# B&R Automation Studio project AS
Automation Studio 4.2.4.149

## Configuration Config1

CPU 5PC800.B945-02, AutomationRuntime A4.26, Build 4.1.2, Vc V4.26.0

### Cpu.per - 5PC800_B945_02/Cpu.per
```iecst
VAR_CONFIG
	gRecCfg AT %M0; (* *)
END_VAR
```

### cncSpindle.mpspindle - 5PC800_B945_02/mapp/cncSpindle.mpspindle
```
Element Spindle_MpLink (Type=mpspindle)
  AxisConfiguration = AxisWithConfiguration
    Axis:
      MeasurementResolution = 0.001
      MovementLimits:
        VelocityPositive = 360000
        VelocityNegative = 360000
        Acceleration = 36000
        Deceleration = 36000
        JerkTime = 0.01
    Drive:
      Controller:
        LoopFilters:
          [0]
          [1]
          [2]
  Alarms = MpAlarmX
```

### deltaCtrl.mpdelta4axis - 5PC800_B945_02/mapp/deltaCtrl.mpdelta4axis
```
Element Delta_MpLink (Type=mpdelta4axis)
  Linking:
    Subnodes:
      JointQ1 = Axis_Delta_Joint_Q1_MpLink
      JointQ2 = Axis_Delta_Joint_Q2_MpLink
      JointQ3 = Axis_Delta_Joint_Q3_MpLink
      Rotary = Axis_Delta_Joint_Q4_MpLink
  Robot:
    Mechanics:
      BasePosition:
        Z = 938.87
      ArmLinkPoint:
        [0]:
          Radius = 200
        [1]:
          Angle = 120
          Radius = 200
        [2]:
          Angle = 240
          Radius = 200
      ArmLength:
        [0]:
          UpperArm = 350
          LowerArm = 800
        [1]:
          UpperArm = 350
          LowerArm = 800
        [2]:
          UpperArm = 350
          LowerArm = 800
      TCPLinkPoint:
        [0]:
          Radius = 45
        [1]:
          Radius = 45
        [2]:
          Radius = 45
    Joint:
      [0]:
        NegativeMoveLimit = -150
        PositiveMoveLimit = 970
        UseTRFLimits = FALSE
      [1]:
        NegativeMoveLimit = -150
        PositiveMoveLimit = 970
        UseTRFLimits = FALSE
      [2]:
        NegativeMoveLimit = -150
        PositiveMoveLimit = 970
        UseTRFLimits = FALSE
    Rotary:
      UseTRFLimits = FALSE
    WorkspaceMonitoring:
      ProtectedBlock:
        [0]
        [1]
        [2]
        [3]
        [4]
      ProtectedHalfSpace:
        [0]
        [1]
        [2]
        [3]
        [4]
  Alarms = MpAlarmX
```

## Configuration Config_MpView

CPU 5PC800.B945-02, AutomationRuntime A4.26, Build 4.1.2, Vc V4.26.0, Safety 0.0

### Arnc0cfg.ncc - 5PC800_B945_02/Motion/Arnc0cfg.ncc
```
NcConfiguration (Version=3.14.3, NcSwId=Arnc0)
  ARNC0CFG_typ:
    sampling_rate = 2000
    cnt_nettrc_rec_drive = 150
    bufsize_sys_trace = 16#00005000
    enable_mp_log = Yes
    tc_nc_man_task = Cyclic #1
    bg_load = 1
    glob_pv_as_ncobject = No
```

### AlarmXCore.mpalarmxcore - 5PC800_B945_02/mapp/AlarmXCore.mpalarmxcore
```
Element MpLink_AlarmControl (Type=mpalarmxcore)
  mapp.AlarmX.Core:
    Mapping:
      [0]:
        Alarm = exampleAlarm
        [0] = Reaction
          Name = exampleReaction
    Default:
      [0] = Reaction
  mapp.AlarmX.Core.Configuration:
    [0]:
      Name = exampleAlarm
      Message = {$alarm/txtExampleAlarm}
      Code = 123456
  mapp.AlarmX.Core.Snippets:
    [0]:
      Key = exampleSnippet
      Value:
        PV = ::AlarmX:loc.val_float
```

### Energy.mpenergycore - 5PC800_B945_02/mapp/Energy.mpenergycore
```
Element Energy_MpLink (Type=mpenergycore)
  Alarms = MpAlarmX
```

### RecCfg.mprecipecsv - 5PC800_B945_02/mapp/RecCfg.mprecipecsv
```
Element Recipe_CSV_MpLink (Type=mprecipecsv)
  mapp.Recipe.Csv:
    Format:
      DecimalMark = .
  Alarms = MpAlarmX
Element Config_CSV_MpLink (Type=mprecipecsv)
  mapp.Recipe.Csv:
    Format:
      DecimalMark = .
  Alarms = MpAlarmX
```

### cncAxes.mpaxisbasic - 5PC800_B945_02/mapp/cncAxes.mpaxisbasic
```
Element Axis_CNC_Z_MpLink (Type=mpaxisbasic)
  AxisConfiguration = AxisWithConfiguration
    Axis:
      MeasurementResolution = 0.001
      SoftwareLimitPositions:
        LowerLimit = -1000
        UpperLimit = 1000
      MovementLimits:
        VelocityPositive = 200
        VelocityNegative = 200
        Acceleration = 500.0
        Deceleration = 500.0
        JerkTime = 0.05
        PositionErrorStopLimit = 1
        VelocityErrorStopLimit = 1
    Drive:
      Transformation:
        ReferenceDistance = 5
      Controller:
        LoopFilters:
          [0]
          [1]
          [2]
  Alarms = MpAlarmX
Element Axis_CNC_Y_MpLink (Type=mpaxisbasic)
  AxisConfiguration = AxisWithConfiguration
    Axis:
      MeasurementResolution = 0.001
      SoftwareLimitPositions:
        LowerLimit = -1000
        UpperLimit = 1000
      MovementLimits:
        VelocityPositive = 200
        VelocityNegative = 200
        Acceleration = 500.0
        Deceleration = 500.0
        JerkTime = 0.05
        PositionErrorStopLimit = 1
        VelocityErrorStopLimit = 1
    Drive:
      Transformation:
        ReferenceDistance = 5
      Controller:
        LoopFilters:
          [0]
          [1]
          [2]
  Alarms = MpAlarmX
Element Axis_CNC_X_MpLink (Type=mpaxisbasic)
  AxisConfiguration = AxisWithConfiguration
    Axis:
      MeasurementResolution = 0.001
      SoftwareLimitPositions:
        LowerLimit = -1000
        UpperLimit = 1000
      MovementLimits:
        VelocityPositive = 200
        VelocityNegative = 200
        Acceleration = 500.0
        Deceleration = 500.0
        JerkTime = 0.05
        PositionErrorStopLimit = 1
        VelocityErrorStopLimit = 1
    Drive:
      Transformation:
        ReferenceDistance = 5
      Controller:
        LoopFilters:
          [0]
          [1]
          [2]
  Alarms = MpAlarmX
```

### deltaTch.mpteachpointui - 5PC800_B945_02/mapp/deltaTch.mpteachpointui
```
Element Teach_MpLink (Type=mpteachpointui)
  TeachPoint:
    Generation:
      UseRapidVelocity = TRUE
  Alarms = MpAlarmX
```

## Configuration Config_Test

### Hardware
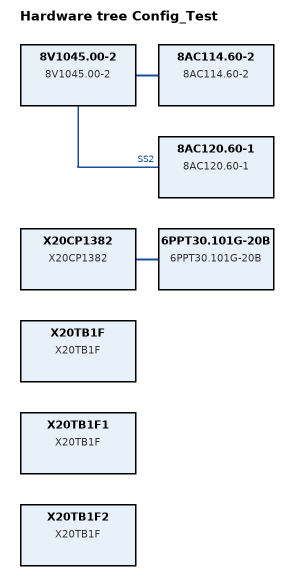
```
6PPT30.101G-20B : 6PPT30.101G-20B v1.1.0.0  [ETH1 -> X20CP1382.IF2 (NodeNumber=1)]
  Terminal = true
  Startmode = 1
  ShowBootlogoVNC = 1
  Mode = Manual
  InternetAddress = 192.168.10.20
  DefaultGateway = 192.168.10.1
  Subnetmask = 255.255.255.0
  Hostname = t30
  Displaybrightness = 75
  PasswordVNC = 
  PasswordCIFS = 
  PasswordService = 
  VncKeyMappingFile = VC\6PPT30.101G-20B.dis
  VncRefreshRate = 200
8AC114.60-2 : 8AC114.60-2 v1.0.0.8  [SS -> 8V1045.00-2.SS1; PLK1 -> X20CP1382.IF3 (NodeNumber=1)]
8AC120.60-1 : 8AC120.60-1 v1.0.0.2  [SS -> 8V1045.00-2.SS2]
8V1045.00-2 : 8V1045.00-2 v1.0.0.2
  SinglePhaseOperation = on
  AxisIsPeriodic_r1 = on
  BothEndSwitchesAreNormallyOpen_r1 = on
  QuickStopIsNormallyOpen_r1 = on
  SupplyVoltage = 200
X20CP1382 : X20CP1382 v1.3.0.0  [X1 -> X1.SL; X2 -> X2.SL; X3 -> X3.SL]
  Module X1 (Type=X1, Virtual=true, Version=1.0.0.0)
    Connection (Connector=SS1, TargetModule=X20TB1F, TargetConnector=SS)
    Connection (Connector=SL, TargetModule=X20CP1382, TargetConnector=X1)
  Module X2 (Type=X2, Virtual=true, Version=1.0.0.0)
    Connection (Connector=SS1, TargetModule=X20TB1F1, TargetConnector=SS)
    Connection (Connector=SL, TargetModule=X20CP1382, TargetConnector=X2)
  Module X3 (Type=X3, Virtual=true, Version=1.0.0.0)
    Connection (Connector=SS1, TargetModule=X20TB1F2, TargetConnector=SS)
    Connection (Connector=SL, TargetModule=X20CP1382, TargetConnector=X3)
  Connector IF2:
    ActivateDevice = 1
    HostName = cp13
    Mode = Manual
    InternetAddress = 192.168.10.10
    SubnetMask = 255.255.255.0
    Vnc1
    VncVcObjectName1 = WSVGA
    VncKeyMappingFile1 = VC\PS2-Keyboard.dis
    VncMaxConnections1 = 2
    VncRefreshRate1 = 100
  Connector IF3:
    CycleTime = 4000
  ConfigurationID = Framework_Config1
  UserPartitionSize = 256
  AutomaticTransferOfUserfiles = on
  ApplicationStorageType = NORMAL
  Simulation = 1
  UserRamSize = 15000
  RemMemSize = 5000
  PermanentPvSize = 2500
  RemanentGlobalPvSize = 1000
  VolatileGlobalPvSize = 350000
  TimerDeviceType = EPLX2X
  TimerDevice = X20CP1382.IF3
  TaskClassIdleTime = 8000
  Cyclic1Duration = 4000
  Cyclic1Tolerance = 0
  Cyclic2Duration = 12000
  Cyclic2Tolerance = 84000
  Cyclic3Duration = 48000
  Cyclic3Tolerance = 48000
  Cyclic4Duration = 100000
  Cyclic4Tolerance = 100000
  Cyclic5Duration = 200000
  Cyclic5Tolerance = 200000
  Cyclic6Duration = 500000
  Cyclic6Tolerance = 500000
  Cyclic7Duration = 1000000
  Cyclic7Tolerance = 1000000
  Cyclic8Duration = 48000
  Cyclic8Tolerance = 30000000
  ActivateOpcUa = 1
  OpcUa_Security_SoftwareCertificates = 
X20TB1F : X20TB1F v1.0.0.0
X20TB1F1 : X20TB1F v1.0.0.0
X20TB1F2 : X20TB1F v1.0.0.0
```

### Acp10cfg.ncc - X20CP1382/Motion/Acp10cfg.ncc
```
NcConfiguration (Version=3.16.2, NcSwId=Acp10)
  ACP10CF1_typ:
    cnt_nettrc_rec_drive = 150
    bufsize_trace_upload = 1200
    tc_nc_man_task = Cyclic #1
    glob_pv_as_ncobject = Yes
    ncsys_dl_broadcast = Yes
    ncsys_dl_acp_reset = Yes
    safemc_log_err_to_ax = Yes
    network_init:
      ncsw_init_execute = Yes
      automatic_execute = No
      node_nr_warning = Yes
      net_err_before_ncact = Yes
    nettrc:
      enter_parsecrec = Yes
      enter_ncaction = Yes
      save_ring_startidx = No
    cam_prof_download:
      cam_dat_dl_parallel = No
      tc_cam_dl_parallel = Task class for NC Manager task
    plk_if[0]:
      if_name = IF3
      tc_CycDat_PLCopen = Task class for NC Manager task
      mc_broadcast_extdat = No
```

### Arnc0map.ncm - X20CP1382/Motion/Arnc0map.ncm
```
NcMapping (NcSwId=Arnc0, DisabledNodesAreHidden=False)
  NcObject CNC_Group (Type=ncCNCSYS, Channel=1, AcoposSimulation=Off, InitParameter=CNC_Init, Disabled=FALSE, ModuleDisabled=FALSE)
  NcObject Delta_Group (Type=ncCNCSYS, Channel=2, AcoposSimulation=Off, InitParameter=Delta_Init, Disabled=FALSE, ModuleDisabled=FALSE)
  NcObject CNC3 (Type=ncCNCSYS, Channel=3, AcoposSimulation=Off, Disabled=TRUE, ModuleDisabled=FALSE)
  NcObject CNC4 (Type=ncCNCSYS, Channel=4, AcoposSimulation=Off, Disabled=TRUE, ModuleDisabled=FALSE)
  NcObject CNC5 (Type=ncCNCSYS, Channel=5, AcoposSimulation=Off, Disabled=TRUE, ModuleDisabled=FALSE)
  NcObject CNC6 (Type=ncCNCSYS, Channel=6, AcoposSimulation=Off, Disabled=TRUE, ModuleDisabled=FALSE)
  NcObject CNC7 (Type=ncCNCSYS, Channel=7, AcoposSimulation=Off, Disabled=TRUE, ModuleDisabled=FALSE)
  NcObject CNC8 (Type=ncCNCSYS, Channel=8, AcoposSimulation=Off, Disabled=TRUE, ModuleDisabled=FALSE)
  NcObject CNC9 (Type=ncCNCSYS, Channel=9, AcoposSimulation=Off, Disabled=TRUE, ModuleDisabled=FALSE)
  NcObject CNC10 (Type=ncCNCSYS, Channel=10, AcoposSimulation=Off, Disabled=TRUE, ModuleDisabled=FALSE)
  NcObject CNC11 (Type=ncCNCSYS, Channel=11, AcoposSimulation=Off, Disabled=TRUE, ModuleDisabled=FALSE)
  NcObject CNC12 (Type=ncCNCSYS, Channel=12, AcoposSimulation=Off, Disabled=TRUE, ModuleDisabled=FALSE)
  NcObject CNC13 (Type=ncCNCSYS, Channel=13, AcoposSimulation=Off, Disabled=TRUE, ModuleDisabled=FALSE)
  NcObject CNC14 (Type=ncCNCSYS, Channel=14, AcoposSimulation=Off, Disabled=TRUE, ModuleDisabled=FALSE)
  NcObject CNC15 (Type=ncCNCSYS, Channel=15, AcoposSimulation=Off, Disabled=TRUE, ModuleDisabled=FALSE)
  NcObject CNC16 (Type=ncCNCSYS, Channel=16, AcoposSimulation=Off, Disabled=TRUE, ModuleDisabled=FALSE)
  NcObject CNC17 (Type=ncCNCSYS, Channel=17, AcoposSimulation=Off, Disabled=TRUE, ModuleDisabled=FALSE)
  NcObject CNC18 (Type=ncCNCSYS, Channel=18, AcoposSimulation=Off, Disabled=TRUE, ModuleDisabled=FALSE)
  NcObject CNC19 (Type=ncCNCSYS, Channel=19, AcoposSimulation=Off, Disabled=TRUE, ModuleDisabled=FALSE)
  NcObject CNC20 (Type=ncCNCSYS, Channel=20, AcoposSimulation=Off, Disabled=TRUE, ModuleDisabled=FALSE)
  NcObject CNC21 (Type=ncCNCSYS, Channel=21, AcoposSimulation=Off, Disabled=TRUE, ModuleDisabled=FALSE)
  NcObject CNC22 (Type=ncCNCSYS, Channel=22, AcoposSimulation=Off, Disabled=TRUE, ModuleDisabled=FALSE)
  NcObject CNC23 (Type=ncCNCSYS, Channel=23, AcoposSimulation=Off, Disabled=TRUE, ModuleDisabled=FALSE)
  NcObject CNC24 (Type=ncCNCSYS, Channel=24, AcoposSimulation=Off, Disabled=TRUE, ModuleDisabled=FALSE)
```

### AlarmXHist.mpalarmxhistory - X20CP1382/mapp/AlarmXHist.mpalarmxhistory
```
Element MpLink_AlarmHistory (Type=mpalarmxhistory)
```

### AxisConfig.mpaxisbasic - X20CP1382/mapp/AxisConfig.mpaxisbasic
```
Element Axis_MpLink (Type=mpaxisbasic)
```

### File_Mgmt.mpfilemanagerui - X20CP1382/mapp/File_Mgmt.mpfilemanagerui
```
Element File_Manager_MpLink (Type=mpfilemanagerui)
  Alarms = MpAlarmX
```

## Logical view

Binary libraries used (declarations not repeated): operator, runtime, astime, AsIecCon, brsystem, sys_lib, ArEventLog, DataObj, FileIO, AsArProf, AsMem, ArTextSys, ArUser, AsANSL, AsARCfg, AsArSdm, AsBrMath, AsBrStr, AsBrWStr, AsCont, AsGuard, AsHost, AsICMP, AsIO, AsIOAcc, AsIODiag, AsIOTime, AsFltGen, AsMath, AsOpcUac, AsPciStr, AsSafety, AsXml, standard, AsTCP, AsUDP, dvframe, AsUSB, AsWStr, MpCom 1.40.1, MpAlarmX, MpAudit 1.40.1, vclib, visapi, MpData, MpEnergy 1.40.1, MpFile 1.40.1, MpOee, MpPackML 1.40.1, MpRecipe, MpReport 1.40.1, MpUserX, MpWebXs 1.40.1, vncserv, AsEPL, AsArLog, Acp10_MC, Acp10man 3.16.2, NcGlobal, Acp10par 3.14.3, Acp10sdc 3.16.2, Acp10sim 3.14.3, Arnc0man 3.14.3, Arnc0mx 3.14.3, MpAxis 1.40.1, MpDelta 1.40.1, GmcGrpAPI, GmcArncGrp, GmcManager 0.69.2, TRF_LIB, MTProfile, jgLibC, wbrListSvc, wbrFltUtil, wbrBytUtil, lib5200

### Global.var - Global variables
```iecst
VAR
	gHmiParamTable : hmiParamListTable_typ := (0); (*Machine configuration / parameter settings logic *)
	gAlarms : applicationAlarms_typ := (0);
	gAlarmsFiltered : applicationAlarms_typ := (0);
END_VAR
```

### Variables.var
```iecst
VAR CONSTANT
	svnIsInVCSSytem : STRING[80] := 'not versioned';
	svnURL : STRING[80] := 'http://99.33.108.51/Internal/Template_V2/trunk/Software/Framework';
	svnCompileTime : STRING[80] := '2016/11/22 15:50:28';
	svnPullDate : STRING[80] := '2016/11/22 15:42:08';
	svnContainsModifications : STRING[80] := 'Modified';
	svnRevision : STRING[80] := 'R587';
	svnRange : STRING[80] := '584:587';
END_VAR
```

### template_info.txt
```
VAR CONSTANT
	svnIsInVCSSytem : STRING[80] := '$WCINSVN?versioned:not versioned$';
	svnURL : STRING[80] := '$WCURL$';
	svnCompileTime : STRING[80] := '$WCNOW$';
	svnPullDate : STRING[80] := '$WCDATE$';
	svnContainsModifications : STRING[80] := '$WCMODS?Modified:Not modified$';
	svnRevision : STRING[80] := 'R$WCREV$';
	svnRange : STRING[80] := '$WCRANGE$';
END_VAR
```

### Package Logical/Libraries - Global (BuR) libraries


### Program Logical/Libraries/MAPPSuppor

#### HMIparamList.typ
```iecst
(********************************************************************
 * COPYRIGHT -- piedmont
 ********************************************************************
 * Package: HMI
 * File: HMI.typ
 * Author: goran
 * Created: August 28, 2013
 ********************************************************************
 * Data types of package HMI
 ********************************************************************)
(*########################################################################*)
(*HMI object - PARAMETER LIST - LIMITS*)
(*########################################################################*)
(*########################################################################*)
(*HMI object - PARAMETER LIST*)
(*########################################################################*)

TYPE
	HMITableIndex_enum :
		(
		TABLE_REC_CONTROL := 0,
		TABLE_REC_DISPENSE := 1,
		TABLE_CFG_CONTROL := 2,
		TABLE_CFG_DISPENSE := 3
		);
	hmiTableStatStruct_typ : 	STRUCT
		maxLenDesc : UDINT;
		maxLenName : UDINT;
		Param : UDINT;
		Default : UDINT;
		Min : UDINT;
		Max : UDINT;
		Hide : UDINT;
	END_STRUCT;
	hmiTableStats_typ : 	STRUCT
		Overall : hmiTableStatStruct_typ;
	END_STRUCT;
	PVList_Language_Texts_typ : 	STRUCT
		PVTextLangSpecific : STRING[DEFINE_PAR_NAME_MAXLEN];
		PVDescLangSpecific : STRING[DEFINE_PAR_DESC_MAXLEN];
	END_STRUCT;
	PVListTexts_Info_typ : 	STRUCT
		Str : STRING[DEFINE_PAR_NAME_MAXLEN];
		isValid : BOOL;
		isPV : BOOL;
		isConstant : BOOL;
		Const_Value : REAL;
		PVAdr : {REDUND_UNREPLICABLE} UDINT;
		PVLen : USINT;
		PVDim : USINT;
		PVTyp : UDINT;
		StrLen : UDINT;
	END_STRUCT;
	PVTable_Val_Info_typ : 	STRUCT
		Param : PVListTexts_Info_typ;
		Default : PVListTexts_Info_typ;
		Min : PVListTexts_Info_typ;
		Max : PVListTexts_Info_typ;
		Hide : PVListTexts_Info_typ;
	END_STRUCT;
	PVTableInfo : 	STRUCT
		PVText : ARRAY[0..MAX_IDX_LANGUAGES]OF PVList_Language_Texts_typ;
		Val : PVTable_Val_Info_typ;
		Error : BOOL;
	END_STRUCT;
	HMI_Table_Data_typ : 	STRUCT
		info : ARRAY[0..DEFINE_MAX_TABLE_ENTRIES]OF PVTableInfo;
		Max_Idx_Entries : UDINT;
		Table_Name : STRING[DEFINE_PAR_NAME_MAXLEN];
		NameSpace : STRING[DEFINE_PAR_NAME_MAXLEN];
		Load_OK : BOOL;
	END_STRUCT;
	hmiParamLimits_typ : 	STRUCT
		k_factor : REAL; (*scaling k factor (y=kx + n, where y=dsiplay value, x=plc value)*)
		n_factor : REAL; (*scaling n factor (y=kx + n, where y=dsiplay value, x=plc value)*)
		minValue : REAL; (*min value*)
		maxValue : REAL; (*max value*)
		defaultValue : REAL; (*default value*)
		pEnumText : UDINT; (*ptr to a string of comma delimited enum texts*)
		pEnumVals : UDINT; (*ptr to a string of comma delimited enum values*)
		valueType : UINT; (*type of the paramvalue (0-DINT, 1-REAL, 2-ENUM)*)
	END_STRUCT;
	hmiParamListTable_typ : 	STRUCT
		listHeader : STRING[DEFINE_PAR_NAME_MAXLEN]; (*name of the list (header text)*)
		listIdText : ARRAY[0..DEFINE_MAX_TABLE_ENTRIES]OF STRING[DEFINE_PAR_IDX_MAXLEN]; (*table colum: id-s*)
		listTypeText : ARRAY[0..DEFINE_MAX_TABLE_ENTRIES]OF STRING[DEFINE_PAR_NAME_MAXLEN]; (*table colum: value*)
		listDefaultText : ARRAY[0..DEFINE_MAX_TABLE_ENTRIES]OF STRING[DEFINE_PAR_NAME_MAXLEN]; (*table colum: value*)
		listMinText : ARRAY[0..DEFINE_MAX_TABLE_ENTRIES]OF STRING[DEFINE_PAR_NAME_MAXLEN]; (*table colum: value*)
		listMaxText : ARRAY[0..DEFINE_MAX_TABLE_ENTRIES]OF STRING[DEFINE_PAR_NAME_MAXLEN]; (*table colum: value*)
		listValueText : ARRAY[0..DEFINE_MAX_TABLE_ENTRIES]OF STRING[DEFINE_PAR_NAME_MAXLEN]; (*table colum: value*)
		listName : ARRAY[0..DEFINE_MAX_TABLE_ENTRIES]OF STRING[DEFINE_PAR_NAME_MAXLEN]; (*table colum: name*)
		listDescription : ARRAY[0..DEFINE_MAX_TABLE_ENTRIES]OF STRING[DEFINE_PAR_DESC_MAXLEN]; (*table colum: description*)
		listValuePtr : ARRAY[0..DEFINE_MAX_TABLE_ENTRIES]OF UDINT; (*list of ptrs to parametars*)
		listDecPlaces : ARRAY[0..DEFINE_MAX_TABLE_ENTRIES]OF DINT; (*list of dec places for each parametar*)
		listLimits : ARRAY[0..DEFINE_MAX_TABLE_ENTRIES]OF hmiParamLimits_typ;
		selName : {REDUND_UNREPLICABLE} STRING[DEFINE_PAR_NAME_MAXLEN]; (*name of the currently selected/active parametar*)
		selDescription : STRING[DEFINE_PAR_DESC_MAXLEN]; (*description of the currently selected/active parametar*)
		selValueEnumIndex : UDINT; (*value of the currently selected/active parametar for type enum*)
		selValueEnumIndexMax : UDINT; (*value of the currently selected/active parametar for type enum*)
		selValueREAL : REAL; (*value of the currently selected/active parametar*)
		selValueREALOld : REAL; (*value of the currently selected/active parametar (previous value for change detection*)
		selValueREALMax : REAL; (*max value of the currently selected/active parametar*)
		selValueREALMin : REAL; (*min value of the currently selected/active parametar*)
		selValueREALDefault : REAL; (*default value of the currently selected/active parametar*)
		selValueDecPlaces : DINT; (*default value of the currently selected/active parametar*)
		selValueDINT : DINT; (*value of the currently selected/active parametar*)
		selValueDINTOld : DINT; (*value of the currently selected/active parametar (previous value for change detection*)
		selValueDINTMax : DINT; (*max value of the currently selected/active parametar*)
		selValueDINTMin : DINT; (*min value of the currently selected/active parametar*)
		selValueDINTDefault : DINT; (*default value of the currently selected/active parametar*)
		selValueFormVisible : DINT; (*visibility control of the form / controls for setting parametar value*)
		index : UINT; (*index of the currently selected/active parametar*)
		indexOld : UINT; (*index of the currently selected/active parametar (previous value for change detection)*)
		maxIndex : UINT; (*max index / number of items in the table. Must be less then hmiTableMAXDESCRIPTION!!!*)
		setDefaultRequest : BOOL; (*set default request flag*)
		incDP : USINT;
		decDP : USINT;
	END_STRUCT;
END_TYPE
```

#### bgstring.c
```c
#ifndef _BG_STRING_C
#define _BG_STRING_C

#ifdef WIN32
#include "string.h"
#else
#include <bur/plctypes.h>
#endif
#include "bgstring.h"

/*
File:
bgString.c

About:
------
- implements  additional string manipulation functions

B&R System Dependencies:
------------------------
- B&R system library: libasstring.a
- B&R system header files: asstring.h

History:
--------
09/11/2005
- rectified issue with bgStringListLines() to properly handle zero length
input string

05/08/2005
-first version

Test and example code:
----------------------
- to run this file standalone:
--- enable following code section (remove or comment out #if 0 / #endif)
--- create cyclic object (task) from C Language and add this file
*/

#if 0
#include <bur/plc.h>
#include <bur/plctypes.h>

#define TXT_SIZE 64
_LOCAL char textBuffer1[TXT_SIZE];
_LOCAL char textBuffer2[TXT_SIZE];
_LOCAL int idxResult;
_LOCAL int idxStart;
_LOCAL int idxEnd;

_INIT void Init(void) {

	/*use defaults*/
	idxStart 	= -1;
	idxEnd 		= -1;
	/*start with empty strings*/
	textBuffer1[0] = 0;
	textBuffer2[0] = 0;
}

_CYCLIC void Cyclic(void) {

	idxResult = bgStrFind(textBuffer1, textBuffer2, start, end);

}
#endif

/*End: Example/Test code*/
int bgStrFind(char *s, char *sub, int idxStart, int idxEnd)
{
	int i, j;
	int subLen;
	char *ptrStr;
	char *ptrSub;

	/*exit if null ptrs*/
	if(!s || !sub)
		return -1;

	/*exit if zero strings*/
	if( !(*s) || !(*sub) )
		return -1;

	subLen = strlen(sub);

	/*check starting index: default = -1 -> start @ s[0]*/
	if(idxStart < 0)
		idxStart = 0;

	/*check end index: default = -1 -> end is sLength - subLength*/
	if(idxEnd < 0){
		idxEnd = strlen(s) - subLen;
	}

	/*check if start is beyond the end*/
	if(idxStart > idxEnd)
		return -1;

	/*search for string <sub> within the string <s>*/
	for(i=idxStart; i<=idxEnd; i++)
	{
		ptrStr = s + i;
		ptrSub = sub;

		for(j=0; j<subLen; j++, ptrStr++, ptrSub++)
		{
			if( *ptrStr!= *ptrSub)
				break;
		}

		if( j == subLen)
			return i;
	}

	return -1;
}

/*
bgStrFindEx - has an extra option
option = 0; same as bgStrFind
option = 1; before comparing, both strings are converted to lower case
*/
int bgStrFindEx(char *s, char *sub, int idxStart, int idxEnd, int option)
{
	int i, j;
	int subLen;
	char *ptrStr;
	char *ptrSub;

	/*exit if null ptrs*/
	if(!s || !sub)
		return -1;

	/*exit if zero strings*/
	if( !(*s) || !(*sub) )
		return -1;

	subLen = strlen(sub);

	/*check starting index: default = -1 -> start @ s[0]*/
	if(idxStart < 0)
		idxStart = 0;

	/*check end index: default = -1 -> end is sLength - subLength*/
	if(idxEnd < 0){
		idxEnd = strlen(s) - subLen;
	}

	/*check if start is beyond the end*/
	if(idxStart > idxEnd)
		return -1;

	/*search for string <sub> within the string <s>*/
	for(i=idxStart; i<=idxEnd; i++)
	{
		ptrStr = s + i;
		ptrSub = sub;

		for(j=0; j<subLen; j++, ptrStr++, ptrSub++)
		{
			if(!option){
				if( *ptrStr!= *ptrSub)
					break;
			}else{
				if( bgCharToLowerCase(*ptrStr) != bgCharToLowerCase(*ptrSub) )
					break;
			}
		}

		if( j == subLen)
			return i;
	}

	return -1;
}

int bgStrCpyN(char *dest, char *src, int maxNoOfCharsToCopy)
{
int i;

	/*maxNoOfCharsToCopy-1 - takes into consideration that supplied max
	length is usually the buffer size, 1 char is needed for null termination
	*/
	for(i=0; i<(maxNoOfCharsToCopy-1);i++){
		*(dest+i)=*(src+i);
		if(! (*(src+i) ) )
			break;
	}

	/*if max reached, terminate dest string*/
	if(i >= (maxNoOfCharsToCopy-1))
		*(dest+i)=0;

	/*string termination is not included in the string length*/
	return i;
}

int bgStrTrimCRLF(char *s)
{
int i;
char c;

	for(i=0;i<255;i++){

		c = s[i];

		if( !c )
			break;

		if( (c == 0xa) || (c == 0xd) ){
			s[i] = 0;
			break;
		}
	}

	return i;
}

int bgStrCpyNTrimLeadingSpaces(char *dest, char *src, int maxNoOfCharsToCopy)
{
int i;
int found;
char *srcStart;

	/*look for leading spaces*/
	found = 0;
	for(i=0; i<(maxNoOfCharsToCopy-1);i++){
		if( *(src+i) != ' ' ){
			srcStart = src + i;
			found = 1;
			break;
		}
	}

	if(!found){
	/*src string is all spaces->set destination to empty string*/
		*dest = 0;
		return 0;
	}

	return bgStrCpyN(dest, srcStart, maxNoOfCharsToCopy);
}

/*
copy string, don't go over the size of dest buffer, trim leading / trailing spaces / convert
to lower case
*/
int bgStrCpyNTrimSpcsToLwr(char *dest, char *src, int maxNoOfCharsToCopy)
{
int i;
char* srcStart = src;
char* srcEnd;
int len = strlen(src);

	if( !len )
		return len;

	/*find src start, avoid leading spaces*/
	while(1){
		if( *srcStart != ' ')
			break;

		if( *srcStart == 0)
			return 0;

		srcStart++;
	}

	/*find src end, trim trailing spaces*/
	srcEnd = (char*)(src + len - 1);
	while(1){
		if( *srcEnd != ' ')
			break;

		if( *srcEnd == 0)
			return 0;

		srcEnd--;
	}

	srcEnd++;

	if( srcStart >= srcEnd )
		return 0;

	for(i=0; i<(maxNoOfCharsToCopy-1); i++){
		dest[i] = bgCharToLowerCase(*srcStart);
		srcStart++;
		if(srcStart >= srcEnd){
			i++;
			break;
		}
	}

	dest[i] = 0;
	return i;
}

int bgIsDigit(char c){
	return ((c>='0') && (c<='9')) ? 1 : 0;
}

#if 0
/*
Test for: bgStringListLinesEx()

The xxxxEx functions use externaly supplied buffer space to store result pointers to
lines / words.
Based on the supplied buffer size, functions will calculate max. number of items (char ptr-s)
that may be stored within the given / allocated storage area.
See: pList->itemCountMax

To test it out, create a new cyclic task then use following code!
*/
#include <bur/plc.h>
#include <bur/plctypes.h>

#include "bglib/bgString.h"
#include "bglib/bgString.c"

#include "bglib/bgdebug.h"
#include "bglib/bgringbuffer.c"

_LOCAL bgStringListEx_typ listLines;
_LOCAL bgStringListEx_typ listWords;
_LOCAL char multiLineTextBuffer[256];
_LOCAL int lineCount;
_LOCAL int wordCount;
_LOCAL int test;
_LOCAL char listPtrBuf[128];    /*this is a "free" storage for list ptr-s! use it with caution!*/

_INIT void init()
{
	strcpy(multiLineTextBuffer, "hello world\r\nThis is a test for second line!\r\nThird line is here and there...\r\nLine #4 : right.left dot !\r\n");
	test = 0;
}

_CYCLIC void cyclic()
{
int i, j;

/*
This is just an example on how to use external / user supplied buffer in order to
store line / word lists. Based on the supplied buffer size, functions will calculate
max. number of items that may be stored within the given / allocated storage area.
See: pList->itemCountMax
*/
char* lineListStorage = &listPtrBuf[0];
char* wordListStorage = &listPtrBuf[64];

	if( test ){
		test = 0;

		lineCount = bgStringListLinesEx(&listLines, multiLineTextBuffer, lineListStorage, 64);
		DBG("multiLineTextBuffer has lineCount=%d lines. (same as listLines.itemCount= %d). Lines are:\r\n", lineCount, listLines.itemCount);
		for(i=0; i<listLines.itemCount; i++){
			DBG("Line[%d]->%s\r\n", i, listLines.items[i]);
			wordCount = bgStringSplitLineEx(&listWords, ' ', listLines.items[i], wordListStorage, 64);
				DBG("     Line[%d] has wordCount=%d words. (same as listWords.itemCount= %d). Words are:\r\n", i, wordCount, listWords.itemCount)
			for(j = 0; j<listWords.itemCount; j++)
				DBG("     Word[%d]->%s\r\n", j, listWords.items[j]);
		}
	}
}
#endif
int bgStringListLines(bgStringList_typ * p){
unsigned char *ptrItemStart, *ptrItemEnd;
int	calcItemCount;

/*
	length = strlen( p->src );
*/
	p->itemCount = 0;

	ptrItemStart = p->src;
	ptrItemEnd = p->src;

	if( *ptrItemStart == 0){
		return 0;
	}

/*process the rest; build list of item pointers*/
	calcItemCount 	= 0;
	while( 1 ){
		if( (*ptrItemEnd == 0x0D) || (*ptrItemEnd == 0x0A)){
			*ptrItemEnd = 0;
			p->items[calcItemCount] = ptrItemStart;
			ptrItemEnd++;

			/*check for an additional \r or \n*/
			if( (*ptrItemEnd == 0x0D) || (*ptrItemEnd == 0x0A)){
				ptrItemEnd++;
			}

			ptrItemStart = ptrItemEnd;
			calcItemCount++;

			if(calcItemCount >= BG_STRINGLIST_MAXITEMCOUNT){
				p->itemCount = calcItemCount;
				return -1;
			}

			/*check for an end of the src string*/
			if( (*ptrItemEnd == 0) ){
				p->itemCount = calcItemCount;
				return calcItemCount;
			}
		}else
		if( *ptrItemEnd == 0){
			p->items[calcItemCount] = ptrItemStart;
			calcItemCount++;
			break;
		}else
			ptrItemEnd++;
	}/*while*/

	p->itemCount = calcItemCount;
	return calcItemCount;
}

void bgStringListExMemSet(bgStringListEx_typ *p, char* pAddrListBuffer, int sizeListBuffer)
{
	/*NOTE: we are going to use supplied char buffer as the storage for the array of char ptr-s!*/
    p->items = (unsigned char**)pAddrListBuffer;

	p->itemCountMax = sizeListBuffer / sizeof(char*);
}

int bgStringListLinesEx(bgStringListEx_typ * p, char* pContentBuffer, char* pAddrListBuffer, int sizeListBuffer){
unsigned char *ptrItemStart, *ptrItemEnd;
int	calcItemCount;

    p->src = (unsigned char*)pContentBuffer;

    /*if mem data is defined, use it; otherwise, mem shall have been set using a separate call to xxxExMemSet()*/
    if(pAddrListBuffer && sizeListBuffer)
        bgStringListExMemSet(p, pAddrListBuffer, sizeListBuffer);

	p->itemCount = 0;

	ptrItemStart = p->src;
	ptrItemEnd = p->src;

	if( *ptrItemStart == 0){
		return 0;
	}

/*process the rest; build list of item pointers*/
	calcItemCount 	= 0;
	while( 1 ){
		if( (*ptrItemEnd == 0x0D) || (*ptrItemEnd == 0x0A)){
			*ptrItemEnd = 0;
			p->items[calcItemCount] = ptrItemStart;
			ptrItemEnd++;

			/*check for an additional \r or \n*/
			if( (*ptrItemEnd == 0x0D) || (*ptrItemEnd == 0x0A)){
				ptrItemEnd++;
			}

			ptrItemStart = ptrItemEnd;
			calcItemCount++;

			if(calcItemCount >= p->itemCountMax){
				p->itemCount = calcItemCount;
				return -1;
			}

			/*check for an end of the src string*/
			if( (*ptrItemEnd == 0) ){
				p->itemCount = calcItemCount;
				return calcItemCount;
			}
		}else
		if( *ptrItemEnd == 0){
			p->items[calcItemCount] = ptrItemStart;
			calcItemCount++;
			break;
		}else
			ptrItemEnd++;
	}/*while*/

	p->itemCount = calcItemCount;
	return calcItemCount;
}

#if 0
Example:
(AS: Make a "C" task; add <filename>.c to the task; copy & paste this code)
#######
#include <bur/plc.h>
#include <bur/plctypes.h>

#include "bgString.h"
#include "bgString.c"

#include "bgdebug.h"

_LOCAL bgStringList_typ myList;
_LOCAL bgStringList_typ mySplitList;
_LOCAL char buffer[256];
_LOCAL int lineCount;
_LOCAL int test;

_INIT void init()
{
	strcpy(buffer, "hello world\r\nwhat is new?\r\nthird line\r\nline #4\r\n");
	test = 0;
}

_CYCLIC void cyclic()
{
int i, j;

	if( test ){
		test = 0;
		myList.src = buffer;
		lineCount = bgStringListLines(&myList);

		for(i=0; i<myList.itemCount; i++){
			DBG("Line[%d]->%s\r\n", i, myList.items[i]);

			mySplitList.src = myList.items[i];
			lineCount = bgStringSplitLine(&mySplitList, ' ');
			for(j = 0; j<mySplitList.itemCount; j++)
				DBG("     Word[%d]->%s\r\n", j, mySplitList.items[j]);
		}
	}
}
######
The above code generates following output (debug telnet client):
>Line[0]->hello world
     Word[0]->hello
     Word[1]->world
Line[1]->what is new?
     Word[0]->what
     Word[1]->is
     Word[2]->new?
Line[2]->third line
     Word[0]->third
     Word[1]->line
Line[3]->line #4
     Word[0]->line
     Word[1]->#4

#endif
int bgStringSplitLine(bgStringList_typ * p, char separator){
unsigned char *ptrItemStart, *ptrItemEnd;
int	calcItemCount;

	p->itemCount = 0;

	ptrItemStart = p->src;
	ptrItemEnd = p->src;

/*process the rest; build list of item pointers*/
	calcItemCount 	= 0;
	while( 1 ){
		if( (*ptrItemEnd == separator) ){
			*ptrItemEnd = 0;
			p->items[calcItemCount] = ptrItemStart;
			ptrItemEnd++;

			calcItemCount++;

			/*check for an additional separtor */
			while( (*ptrItemEnd == separator) ){
				ptrItemEnd++;
				if( (*ptrItemEnd == 0) ){
					p->itemCount = calcItemCount;
					return calcItemCount;
				}
			}

			ptrItemStart = ptrItemEnd;

			if(calcItemCount >= BG_STRINGLIST_MAXITEMCOUNT){
				p->itemCount = calcItemCount;
				return -1;
			}

			/*check for an end of the src string*/
			if( (*ptrItemEnd == 0) ){
				p->itemCount = calcItemCount;
				return calcItemCount;
			}
		}else
		if( *ptrItemEnd == 0){
			p->items[calcItemCount] = ptrItemStart;
			calcItemCount++;
			break;
		}else
			ptrItemEnd++;
	}/*while*/

	p->itemCount = calcItemCount;
	return calcItemCount;
}

int bgStringSplitLineEx(bgStringListEx_typ * p, char separator, char* pLineBuffer, char* pAddrListBuffer, int sizeListBuffer){
unsigned char *ptrItemStart, *ptrItemEnd;
int	calcItemCount;

    p->src = (unsigned char*)pLineBuffer;

    /*if mem data is defined, use it; otherwise, mem shall have been set using a separate call to xxxExMemSet()*/
    if(pAddrListBuffer && sizeListBuffer)
        bgStringListExMemSet(p, pAddrListBuffer, sizeListBuffer);

	p->itemCount = 0;

	ptrItemStart = p->src;
	ptrItemEnd = p->src;

/*process the rest; build list of item pointers*/
	calcItemCount 	= 0;
	while( 1 ){
		if( (*ptrItemEnd == separator) ){
			*ptrItemEnd = 0;
			p->items[calcItemCount] = ptrItemStart;
			ptrItemEnd++;

			calcItemCount++;

			/*check for an additional separtor */
			while( (*ptrItemEnd == separator) ){
				ptrItemEnd++;
				if( (*ptrItemEnd == 0) ){
					p->itemCount = calcItemCount;
					return calcItemCount;
				}
			}

			ptrItemStart = ptrItemEnd;

			if(calcItemCount >= p->itemCountMax){
				p->itemCount = calcItemCount;
				return -1;
			}

			/*check for an end of the src string*/
			if( (*ptrItemEnd == 0) ){
				p->itemCount = calcItemCount;
				return calcItemCount;
			}
		}else
		if( *ptrItemEnd == 0){
			p->items[calcItemCount] = ptrItemStart;
			calcItemCount++;
			break;
		}else
			ptrItemEnd++;
	}/*while*/

	p->itemCount = calcItemCount;
	return calcItemCount;
}

char *bgStringLower(char *s)
{
int i;
char c;

	for(i=0;i<255;i++){

		c = s[i];

		if( !c )
			break;

		if( (c >= 'A') && (c <= 'Z') ){
			s[i] = c - 'A' + 'a';
		}
	}

	return s;
}

char bgCharToLowerCase(char c)
{
char charLowerCase = c;

	if( (c >= 'A') && (c <= 'Z') ){
		charLowerCase = c - 'A' + 'a';
	}

	return charLowerCase;
}

char *bgStringUpper(char *s)
{
int i;
char c;

	for(i=0;i<255;i++){

		c = s[i];

		if( !c )
			break;

		if( (c >= 'a') && (c <= 'z') ){
			s[i] = c - 'a' + 'A';
		}
	}

	return s;
}

int bgStringIsMatch(char *s1, char *s2, int minChrCount)
{
	if( !strcmp(s1, s2) ){
		return 1;
	}else
		return 0;

}

int bgIsNumber_uint(char *s)
{
int i;
char c;

	/*limit execution to 255: don't want cycle time violation due to wrong ptr*/
	for(i=0;i<255;i++){

		c = s[i];

		/*end of valid input string?*/
		if( !c && i)
			return 1;

		/*zero input string?*/
		if( !c && !i)
			return 0;

		/*check if digit or space*/
		if( !bgIsDigit(c) && (c != ' '))
			return 0;
	}

	return 0;
}

int bgIsNumber_int(char *s)
{
int i;
char c;

	/*limit execution to 255: don't want cycle time violation due to wrong ptr*/
	for(i=0;i<255;i++){

		c = s[i];

		/*end of valid input string?*/
		if( !c && i)
			return 1;

		/*zero input string?*/
		if( !c && !i)
			return 0;

		/*check if digit or space*/
		if( !bgIsDigit(c) && (c != ' ') && (c != '-')  && (c != '+'))
			return 0;
	}

	return 0;
}

int bgAsciiToUint(char *src, unsigned int *dst)
{

unsigned int value;

	if( !bgIsNumber_uint(src) )
		return 0;

#ifdef WIN32
	/*TODO!!!*/
	value = 0;
#else
	value = atoi((UDINT)src);
#endif

	*dst = value;

	return 1;
}

int bgAsciiToInt(char *src, unsigned int *dst)
{

unsigned int value;

	if( !bgIsNumber_int(src) )
		return 0;

#ifdef WIN32
	/*TODO!!!*/
	value = 0;
#else
	value = atoi((UDINT)src);
#endif
	*dst = value;

	return 1;
}

int bgStrCopyFromTo(char* src, int srcStartPosition, int srcEndPosition, char* dest)
{
/*
-copy part of the memory from the section of src (from srcStartPosition to srcEndPosition) to dest
-srcEndPosition is not included in the copy (last copied byte position is srcEndPosition-1)
-length of the copied string is (srcEndPosition - srcStartPosition)
Example:
src="01234567890"
srcStartPosition=3
srcEndPosition=7

dest="3456"

return value: number of bytes copied (i.e. length of the dest string)
*/
int size = 0;
int i;

	if( srcEndPosition >= srcStartPosition )
		size = srcEndPosition - srcStartPosition;

	/*do memcopy! end position char is not included in the copy!*/
	for(i=0; i<size; i++)
		dest[i] = src[srcStartPosition + i];

	/*terminate string*/
	dest[size] = 0;

	return size;
}

int bgStrFindEOL(char* src, int startPosition)
{
/*
- search supplied c string "src" (zero terminated!!!) for the eof
- start search at startPosition and look for the first '\n'
- return:
-1 		- EOF (\n) not found
>=0		- EOF position
*/
int position = startPosition;
int i = 0;

	while(1){
		/*end of line?*/
		if( src[position] == '\n' ){
			/*if \r preceeds \n, dec EOL position by 1*/
			if( position && (src[position-1] == '\r') )
				position--;

		 	return position;
		}

 		/*end of string?*/
		if( src[position] == 0 ) return -1;

		/*prevent endless loop*/
		if( ++i >= 4096 ) return -1;

		position++;
	}

	return -1;
}

#endif
/*EOF*/
```

#### hmiTableFBK_typ.c
```c
/// IAUTOMATION CONFIDENTIAL
/// Unpublished Copyright (c) 2016 iAutomation, All Rights Reserved.
///
/// NOTICE:  All information contained herein is, and remains the property of iAutomation. The intellectual and technical concepts contained
/// herein are proprietary to iAutomation and may be covered by U.S. and Foreign Patents, patents in process, and are protected by trade secret or copyright law.
/// Dissemination of this information or reproduction of this material is strictly forbidden unless prior written permission is obtained
/// from iAutomation.  Access to the source code contained herein is hereby forbidden to anyone except current iAutomation employees, managers or contractors who have executed
/// Confidentiality and Non-disclosure agreements explicitly covering such access.
///
/// The copyright notice above does not evidence any actual or intended publication or disclosure  of  this source code, which includes
/// information that is confidential and/or proprietary, and is a trade secret, of  iAutomation.   ANY REPRODUCTION, MODIFICATION, DISTRIBUTION, PUBLIC  PERFORMANCE,
/// OR PUBLIC DISPLAY OF OR THROUGH USE  OF THIS  SOURCE CODE  WITHOUT  THE EXPRESS WRITTEN CONSENT OF COMPANY IS STRICTLY PROHIBITED, AND IN VIOLATION OF APPLICABLE
/// LAWS AND INTERNATIONAL TREATIES.  THE RECEIPT OR POSSESSION OF  THIS SOURCE CODE AND/OR RELATED INFORMATION DOES NOT CONVEY OR IMPLY ANY RIGHTS
/// TO REPRODUCE, DISCLOSE OR DISTRIBUTE ITS CONTENTS, OR TO MANUFACTURE, USE, OR SELL ANYTHING THAT IT  MAY DESCRIBE, IN WHOLE OR IN PART.
///
/// Programmer: John C. Glisson
/// Date: 20. October 2016

#include <bur/plctypes.h>
#ifdef __cplusplus
	extern "C"
	{
#endif
	#include "MAPPSuppor.h"
#ifdef __cplusplus
	};
#endif

#include "hmiParamList.h"
#include "ArTextSys.h"

static void Update_Stats_Table(UDINT * pMaxVal, char * pText, UDINT * pOverallMaxVal){
	UDINT TextLen = 0;

	TextLen = brsstrlen((UDINT) pText);

	if(*pMaxVal < TextLen){
		*pMaxVal = TextLen;
	}
	if(*pOverallMaxVal < TextLen){
		*pOverallMaxVal = TextLen;
	}
	return;
}

static DINT writeText(char * pNameSpace, char * pText, char * pLangCode, char * pParName, UDINT Buffer_Size, UDINT * pTextLen){
	STRING Buffer[Buffer_Size];
	ArTextSysGetText_typ FBK;
	FBK.Namespace = (UDINT) pNameSpace;
	FBK.SearchMode = arTEXTSYS_SEARCH_LANGUAGE_ONLY;
	FBK.TextID = (UDINT) pText;
	brsstrcpy((UDINT) &FBK.LanguageCode, (UDINT) pLangCode);
	FBK.TextBuffer =(UDINT) &Buffer;
	FBK.TextBufferSize = Buffer_Size;

	FBK.Execute = 0;
	ArTextSysGetText(&FBK);
	FBK.Execute = 1;
	ArTextSysGetText(&FBK);

	if(FBK.StatusID == 0){
		brsstrcpy((UDINT) pParName, (UDINT) &Buffer);
		*pTextLen = brsstrlen((UDINT) &Buffer);
	}else{
		brsstrcpy((UDINT) pParName,(UDINT)  &"Err");
	}
	return FBK.StatusID;
}

static DINT Get_PV_Table_Item_Info(char * pNameSpace, char * pTextID, char * pLangCode, PVListTexts_Info_typ * p){
	DINT status = 0;

	status = writeText(pNameSpace,pTextID,pLangCode,(char *) &p->Str, DEFINE_PAR_NAME_MAXLEN, &p->StrLen);

	if(status==0){
		p->isValid = 1;
	}else{
		p->isValid = 0;
		return status;
	}

	status = PV_xgetadr((UDINT) &p->Str,(UDINT) &p->PVAdr,(UDINT) &p->PVLen);

	if(status==0){
		p->isPV = 1;
		p->isConstant = 0;
	}else{
		p->isPV = 0;
		p->isConstant = 1;
		p->Const_Value = brsatof((UDINT) &p->Str);
		return status;
	}

	status = PV_ninfo((UDINT) &p->Str,(UDINT) &p->PVTyp,(UDINT) &p->PVLen,(UDINT) &p->PVDim);
	return status;
}

static void GetPVTableInfo(char * pNameSpace, UDINT pvTableIdx, PVTableInfo * p, BOOL * pErrorFlag){
	char strPVID[DEFINE_PAR_NAME_MAXLEN] = "PV.";
	char strPVIdx[DEFINE_PAR_IDX_MAXLEN];
	DINT status = 0;

	brsitoa(pvTableIdx,(UDINT)  &strPVIdx);
	brsstrcat((UDINT) &strPVID, (UDINT) &strPVIdx);

	status = Get_PV_Table_Item_Info(pNameSpace,		(char *) &strPVID,		(char *) &DEFINE_LANGUAGE_STRINGS[DEFINE_INDEX_TEXTTABLE_PV], 		&p->Val.Param);
	status = Get_PV_Table_Item_Info(pNameSpace,		(char *) &strPVID,		(char *) &DEFINE_LANGUAGE_STRINGS[DEFINE_INDEX_TEXTTABLE_MIN], 		&p->Val.Min);
	status = Get_PV_Table_Item_Info(pNameSpace,		(char *) &strPVID,		(char *) &DEFINE_LANGUAGE_STRINGS[DEFINE_INDEX_TEXTTABLE_MAX], 		&p->Val.Max);
	status = Get_PV_Table_Item_Info(pNameSpace,		(char *) &strPVID,		(char *) &DEFINE_LANGUAGE_STRINGS[DEFINE_INDEX_TEXTTABLE_DEFAULT], 	&p->Val.Default);
	status = Get_PV_Table_Item_Info(pNameSpace,		(char *) &strPVID,		(char *) &DEFINE_LANGUAGE_STRINGS[DEFINE_INDEX_TEXTTABLE_HIDE], 	&p->Val.Hide);
	return;
}

static void GetPVNameInfo(char * pNameSpace, UDINT idxLanguage, UDINT idxPV, char * pParName, char * pParDesc, BOOL * pErrorFlag){
	ArTextSysLanguageCodeType strTmpLang;
	brsstrcpy((UDINT) &strTmpLang, (UDINT) &DEFINE_LANGUAGE_STRINGS[idxLanguage]);
	char strPVName[DEFINE_PAR_NAME_MAXLEN] = "Title.";
	char strPVDesc[DEFINE_PAR_DESC_MAXLEN] = "Desc.";
	char strPVIdx[DEFINE_PAR_IDX_MAXLEN];
	brsitoa((DINT) idxPV, (UDINT) &strPVIdx);
	brsstrcat((UDINT) &strPVName, (UDINT) &strPVIdx);
	brsstrcat((UDINT) &strPVDesc, (UDINT) &strPVIdx);
	UDINT TextLen = 0;

	writeText(pNameSpace, (char *) &strPVName, (char *) &strTmpLang, pParName, DEFINE_PAR_NAME_MAXLEN, &TextLen);
	writeText(pNameSpace, (char *) &strPVDesc, (char *) &strTmpLang, pParDesc, DEFINE_PAR_DESC_MAXLEN, &TextLen);
}

void hmiTableFBK_typ(struct hmiTableFBK_typ* p)
{
	//Really going to try hard to do this all in one cycle.
	UDINT ii_entries=0;
	UDINT ii_languages=0;

	BOOL flagError = 0;

	STRING LogString[DEFINE_LOGSTRING_LEN];

	brsstrcpy((UDINT) &p->hmiStruct.Table_Name,(UDINT)  &p->tableName);
	brsstrcpy((UDINT) &p->hmiStruct.NameSpace,(UDINT)  &p->nameSpace);

	for(ii_entries = 0; ii_entries <= DEFINE_MAX_TABLE_ENTRIES; ii_entries++){
		GetPVTableInfo(p->nameSpace, ii_entries, &p->hmiStruct.info[ii_entries], &flagError);

		if(p->hmiStruct.info[ii_entries].Val.Param.PVAdr == 0){//If there isn't a PV at that index, return from the function...
			p->hmiStruct.Max_Idx_Entries = ii_entries - 1;
			p->hmiStruct.Load_OK = (flagError == 0);

			wbrsnprintf((char *) &LogString, DEFINE_LOGSTRING_LEN, "TableInfo:<Table=%s><Count=%d><err=%d>", &p->tableName, ii_entries, (UDINT) flagError);
			requestMessageToLog((char *) &LogString, p->Logbook, arlogLEVEL_INFO, 50000, 0, 0);

			return;
		}//...Otherwise load its texts

		wbrsnprintf((char *) &LogString, DEFINE_LOGSTRING_LEN, "TableItem:<PVName=%s><Def=%s><Min=%s><Max=%s>", &p->hmiStruct.info[ii_entries].Val.Param.Str, &p->hmiStruct.info[ii_entries].Val.Default.Str, &p->hmiStruct.info[ii_entries].Val.Min.Str, &p->hmiStruct.info[ii_entries].Val.Max.Str);
		requestMessageToLog((char *) &LogString, p->Logbook, arlogLEVEL_INFO, 50000, 0, 0);

		Update_Stats_Table(&p->TableStats.Param,(char *) &p->hmiStruct.info[ii_entries].Val.Param.Str, &p->pOverallStats->Param);
		Update_Stats_Table(&p->TableStats.Default,(char *) &p->hmiStruct.info[ii_entries].Val.Default.Str, &p->pOverallStats->Default);
		Update_Stats_Table(&p->TableStats.Min,(char *) &p->hmiStruct.info[ii_entries].Val.Min.Str, &p->pOverallStats->Min);
		Update_Stats_Table(&p->TableStats.Max,(char *) &p->hmiStruct.info[ii_entries].Val.Max.Str, &p->pOverallStats->Max);
		Update_Stats_Table(&p->TableStats.Hide,(char *) &p->hmiStruct.info[ii_entries].Val.Hide.Str, &p->pOverallStats->Hide);

		for(ii_languages = 0; ii_languages <= MAX_IDX_LANGUAGES; ii_languages++){
			GetPVNameInfo((char *) &p->nameSpace, ii_languages, ii_entries,(char *) &p->hmiStruct.info[ii_entries].PVText[ii_languages].PVTextLangSpecific,(char *)  &p->hmiStruct.info[ii_entries].PVText[ii_languages].PVDescLangSpecific, &flagError);

			Update_Stats_Table(&p->TableStats.maxLenDesc,(char *) &p->hmiStruct.info[ii_entries].PVText[ii_languages].PVDescLangSpecific, &p->pOverallStats->maxLenDesc);
			Update_Stats_Table(&p->TableStats.maxLenName,(char *) &p->hmiStruct.info[ii_entries].PVText[ii_languages].PVTextLangSpecific, &p->pOverallStats->maxLenName);
		}
	}
}
```

- Library Logical/UserLibraries/jgLibs/VA_Setup (ANSIC, version 0.00.0) (no source held here)

- Library Logical/UserLibraries/jgLibs/jgUtils (ANSIC) (no source held here)

### wbrServices.typ - Package data types
```iecst
(*** /*****************************************************************
 * \copyright -- Piedmont Automation
 ********************************************************************
 * Program : wbrServices
 * \file :   wbrServices.typ
 * \author : Blanton Radford
 * \date Created: July 17, 2015
 ********************************************************************
 * Data types of package wbrServices
 ***************************************************************/ *****)

TYPE
	wbrSvc_AsFBStatus_enum :
		(
		wbrSvc_AsFBStatus_SUCCESS := 0,
		wbrSvc_AsFBStatus_NOT_ENABLED := 65534,
		wbrSvc_AsFBStatus_BUSY
		);
	wbrSvcBool_enum :
		(
		NO := 0,
		YES,
		OFF := 0,
		ON,
		STOP := 0,
		START,
		UNCHECK := 0,
		CHECK
		);
	cfgFileInfo_typ : 	STRUCT
		timestamp : STRING[63];
		path : STRING[127];
		machineNumber : UDINT;
		machineName : STRING[31];
	END_STRUCT;
	cfgCompileVersionInfo_typ : 	STRUCT
		projVersion : STRING[63];
		AR_Version : STRING[15];
		AS_config : STRING[63];
		AS_configID : STRING[127];
		AS_build : STRING[63];
		date : STRING[31];
		AS_version : STRING[63];
		user : STRING[63];
		company : STRING[63];
		info : STRING[63];
	END_STRUCT;
END_TYPE

(*wbrUSBService types*)

TYPE
	wbrUSBSvcNodeList_enum :
		(
		wbrusbLAST_NODE := 7,
		wbrusbNUM_NODES
		);
	wbrUSBSvcNodeList_typ : 	STRUCT
		listCurr : {REDUND_UNREPLICABLE} ARRAY[0..wbrusbLAST_NODE]OF UDINT;
		listPrev : {REDUND_UNREPLICABLE} ARRAY[0..wbrusbLAST_NODE]OF UDINT;
		newNodeDetected : {REDUND_UNREPLICABLE} BOOL;
		nodeChangeDetected : {REDUND_UNREPLICABLE} BOOL;
		fb : {REDUND_UNREPLICABLE} UsbNodeListGet;
	END_STRUCT;
	wbrUSBSvcStringDescriptor_typ : 	STRUCT
		isWorking : {REDUND_UNREPLICABLE} BOOL;
		fb : {REDUND_UNREPLICABLE} UsbDescriptorGet;
		descriptor : usbStringDescr_typ;
		descContainer : WSTRING[63] := "";
	END_STRUCT;
	wbrUSBSvcNodeData_typ : 	STRUCT
		isNew : {REDUND_UNREPLICABLE} BOOL;
		isActive : {REDUND_UNREPLICABLE} BOOL;
		isWorking : {REDUND_UNREPLICABLE} BOOL;
		isReady : {REDUND_UNREPLICABLE} BOOL;
		deviceData : usbNode_typ;
		deviceDescriptor : usbDeviceDescr_typ;
		string : ARRAY[0..3]OF wbrUSBSvcStringDescriptor_typ;
		fbGetNode : {REDUND_UNREPLICABLE} UsbNodeGet;
		fbGetDescDev : {REDUND_UNREPLICABLE} UsbDescriptorGet;
		fbMonStorageReady : {REDUND_UNREPLICABLE} UsbMsDeviceReady;
	END_STRUCT;
	wbrUSBService_typ : 	STRUCT
		list : {REDUND_UNREPLICABLE} wbrUSBSvcNodeList_typ;
		node : {REDUND_UNREPLICABLE} ARRAY[0..wbrusbLAST_NODE]OF wbrUSBSvcNodeData_typ;
		nextNodeIdx : {REDUND_UNREPLICABLE} USINT;
	END_STRUCT;
	wbrUSBServiceIF_typ : 	STRUCT
		isReady : {REDUND_UNREPLICABLE} BOOL;
		isFileIODevice : {REDUND_UNREPLICABLE} BOOL; (*Can read and write files on device*)
		fileIODeviceParam : STRING[127] := '---'; (*FileIO device parameter string*)
	END_STRUCT;
END_TYPE
```

### Library Logical/UserLibraries/wbrServices/wbrsprintf (ANSIC) - Writes user-formatted output to a string

#### wbrsprintf.c
```c
/*!
 ********************************************************************
### Library : wbrsprintf
 *  Package : WBRServices
 * \file :   wbrsprintf.c
 * \author : Blanton Radford, Wes Buchanan (B&R), others
 * \date Created: Approximately 2013
 * \copyright -- Piedmont Automation
 *******************************************************************
 * \brief Header file for snprintf functions.
          Use of sprintf functions discouraged as snprintf is guaranteed to
          stop writing once buf_size is filled.
          Write a printf-formatted string to memory at "line"
 ********************************************************************/

#include <stdarg.h>
#include <stdio.h>
#include <limits.h>

#include "wbrsprintf.h"

int __ofmt(FILE *stream, char *line, int buf_size,
                                     const char *format, va_list ap);

int wbrvsprintf(char *s, const char *fmt, va_list ap)
{
  return __ofmt(0, s, INT_MAX, fmt, ap);
}

int wbrvsnprintf(char *s, int buf_size, const char *fmt, va_list ap)
{
  return __ofmt(0, s, buf_size, fmt, ap);
}

int wbrsprintf(char *s, const char *fmt, ...)
{
 int num;
 va_list ap;

  va_start(ap, fmt);
  num = wbrvsprintf(s, fmt, ap);
  va_end(ap);
  return num;
}

int wbrsnprintf(char *s, int buf_size, const char *fmt, ...)
{
 int num;
 va_list ap;

  va_start(ap, fmt);
  num = wbrvsnprintf(s, buf_size, fmt, ap);
  va_end(ap);
  return num;
}
```

### Library Logical/UserLibraries/wbrServices/wbrMemSvc (ANSIC) - Allocate heap memory using AsMem
Depends on: AsMem

#### wbrMemSvc.c
```c
/********************************************************************
 * \copyright -- Piedmont Automation
 ********************************************************************
 * Program : wbrMemSvc
 * \file :   wbrMemSvc.c
 * \author : Blanton Radford
 * \date Created: April 14, 2016
 ******************************************************************* /
 * Implementation of library wbrListSvc
 ********************************************************************/

#include "wbrMemSvc.h"

AsMemPartAllocClear_typ   allocate;
AsMemPartFree_typ         freeMem;
AsMemPartRealloc_typ      reAllocate;
AsMemPartInfo_typ         memInfo;

/*! \todo
*/
UDINT memSvcAllocate(UDINT size)
{
  allocate.len=     size;
  AsMemPartAllocClear(&allocate);
  if(allocate.status == 0)  return  allocate.mem;

  //! \todo   handle errors
  return  0;
}

/*! \brief Init-SP for AsMem heap memory and linked list services
    \warning   This init must be called in the first Init-SP in TC#1
*/
BOOL initMemSvc(UDINT partitionSize)
{
 AsMemPartCreate_typ  getMem;

  getMem.ident= 0;    //  Init to zero for return value - see below

  getMem.enable=
      allocate.enable=
      freeMem.enable=
      reAllocate.enable=
      memInfo.enable=         1;

  getMem.len=     partitionSize;

  AsMemPartCreate(&getMem);

  allocate.ident=
      freeMem.ident=
      reAllocate.ident=
      memInfo.ident=          getMem.ident;

  // return  (BOOL)allocate.ident;    //  WBR:  appears to cause an illegal bool value
  return  allocate.ident != 0;
}

/*! \brief    Frees a block of heap memory

    \pre      \todo
    \warning  \todo

*/
UINT  memSvcFree(UDINT block)
{
  if(!block)
  {
    //! \todo   report null address
    return  0xAAAA;
  }

  freeMem.mem=  block;
  AsMemPartFree(&freeMem);

  if(freeMem.status != 0)
  {
    //!   \todo   possibly loop to try again n times?
    //!   \todo   handle error, flag address for later memory cleanup
  }

  return  freeMem.status;
}

/*! \brief    Returns size of the largest available memory block

    \pre      \todo
    \warning  \todo
    \todo

**/
UDINT memSvcGetMemInfo(wbrMemService_typ * m)
{
  AsMemPartInfo(&memInfo);

  m->status.alloc.status= allocate.status;
  m->status.free.status=  freeMem.status;

  return   memInfo.maxBlockSizeFree;
}
```

### Library Logical/UserLibraries/wbrServices/wbrLogSvc (ANSIC) - Logging to logbooks, other logs todo
Depends on: AsArLog, wbrListSvc, wbrsprintf, ArEventLog

#### wbrLogSvc.c
```c
/********************************************************************
 * \copyright -- Piedmont Automation
 ********************************************************************
 * Program : wbrLogSvc
 * \file :   wbrLogSvc.c
 * \author : Blanton Radford
 * \date Created: May 07, 2015
 ******************************************************************* /
 * Implementation of library wbrLogSvc
 ********************************************************************/

#include "wbrLogSvc.h"

linkedList_typ    *   logList;

wbrLogService_typ *   lsvc;

wbrLogServiceEventLog_typ   sysUserEventLog     //!< Sets up struct data for managing the system user logbook
                          , genericLog
                          ;
wbrLogServiceEventLogEventID_typ  eventID
                                ;

/** Function info
    These functions wrap around multiple instances of AsArLogWrite() in an
array format to implement a LIFO for handling multiple, rapid requests
for entries to the same log module.
    requestMessageToLog() should only be called once for each message to be
inserted. Then, writeMessagesToLog() will continue calling the
appropriate AsArLogWrite() FB instance until the message is written to
the log module (i.e. status == 0). It is possible that the message will
be written to the log on the first call, and so subsequent calls to
writeMessagesToLog() will not be necessary in every case. The busy bit
is be used to control whether or not writeMessagesToLog() needs to be
called.  See
    The entries are (believed to be) timestamped as the original calls are
made to insert them. Therefore the order of the function calls to the
individual FB instances to handle multiple busy statuses is not
important.

 \todo :
- find out why last log entry repeats sometimes rather than printing the entries
  in their proper order. Possible remedies include:
  - (ironically) improve the logging for this service for better debgging
  - delete requested node immediately if status == 0
  - declare new entries on the func stack and only add to list (i.e. copy the fb
    to a list fb) if status == FFFF. Not sure if copying FBs this way will work.
  I believe this is fixed.  Was caused by stack mem being destroyed.  See
    declaration of variable called 'node' in code below.
**/

/*————————————————————————————————————————————————————————————————————————————*/
/*! \brief \b Utility to decode an EventID
    \pre

rtyp  ƒ(x)—————————¬
              ———————————————————————————————————argument   comments————————•••™  */

DINT  decodeEventID(
              DINT                                eventID   //!
            , wbrLogServiceEventLogEventID_typ *  decoded
            )
{
  decoded->code=      (UINT)eventID;
  decoded->facility=  (UINT)(0x0FFF & (eventID >> 16));
  decoded->customer=  (BOOL)(0x0001 & (eventID >> 29));
  decoded->severity= (USINT)(0x0003 & (eventID >> 30));

  return 0;
}
/*————————————————————————————————————————————————————————————————————————————*/

/*————————————————————————————————————————————————————————————————————————————*/
/*! \brief Get last RecordID in logbook
    \pre

rtyp    �(x)뿓뿓뿓뿓뿓뿓뿓뿓뿬  뿓뿓뿓뿓뿓뿓argument comments뿓뿓뿓뿓뿓뿓뿓뿑븬�  */

UDINT   logSvcGetLastRecordID(

          wbrLogServiceEventLog_typ * logInfo       //!< see type for details
        )
{
 static ArEventLogGetLatestRecordID_typ fb;

  fb.Ident= logInfo->access.ident;
  fb.Execute= 1;
  ArEventLogGetLatestRecordID(&fb);

  logInfo->read.oRecordID=  fb.RecordID;

  fb.Execute= 0;
  ArEventLogGetLatestRecordID(&fb);

  return logInfo->read.oRecordID;
}
/*————————————————————————————————————————————————————————————————————————————*/

/*————————————————————————————————————————————————————————————————————————————*/
/*! \brief Get last RecordID output from write
    \pre

rtyp    �(x)뿓뿓뿓뿓뿓뿓뿓뿓뿓뿓뿓뿬  뿓뿓뿓argument comments뿓뿓뿓뿓뿓뿓뿓뿑븬�  */

UDINT    logSvcGetLastWriteRecordID(

          wbrLogServiceEventLog_typ * logInfo       //!< see type for details
        )
{
  return logInfo->write.oRecordID= genericLog.write.oRecordID;
}
/*————————————————————————————————————————————————————————————————————————————*/

/*————————————————————————————————————————————————————————————————————————————*/
/*! \brief Get info about an event logbook
    \pre

rtyp    �(x)뿓뿓뿓뿓뿓뿬  뿓뿓뿓뿓뿓뿓뿓뿓뿓argument comments뿓뿓뿓뿓뿓뿓뿓뿑븬�  */

DINT    getEventLogInfo(

          wbrLogServiceEventLog_typ * logInfo       //!< see type for details
        )
{
 static ArEventLogGetIdent_typ fb;   //  Maybe there will be other info in the future, similar to AsArLogGetInfo()?

  wbrsnprintf(fb.Name, sizeof(fb.Name), logInfo->access.name);

  fb.Execute= 1;
  ArEventLogGetIdent(&fb);

  logInfo->access.ident=  0;
  if(!(logInfo->error= fb.Error))   logInfo->access.ident= fb.Ident;

  logInfo->done=    fb.Done;
  logInfo->status=  fb.StatusID;

  fb.Execute= 0;
  ArEventLogGetIdent(&fb);      //  Clear the fb for next use

  return  logInfo->status;
}
/*————————————————————————————————————————————————————————————————————————————*/

/*————————————————————————————————————————————————————————————————————————————*/
/*! \brief For debugging the log list
*
rtyp              �(x)뿓뿓뿓�  뿓뿓뿓뿓뿓뿓뾞rgument comments뿓뿓뿓뿓뿓뿓뿓뿑븬�  */

linkedList_typ *  getLogList()
{
  return  logList;
}
/*————————————————————————————————————————————————————————————————————————————*/

/*————————————————————————————————————————————————————————————————————————————*/
/*! \brief  Copies log list to pv struct for debugging/monitoring

rtyp    �(x)뿓뿓뿓뿓뿓뿓뿬  뿓뿓뿓뿓뿓뿓뿓뿓argument comments뿓뿓뿓뿓뿓뿓뿓뿑븬�  */

UDINT   getLogServiceData()
{
  // lsvc->list= *(getLogList());
  lsvc->list= *logList;

  return  (UDINT)lsvc;
}

/*————————————————————————————————————————————————————————————————————————————*/

/*————————————————————————————————————————————————————————————————————————————*/
/*! \brief  Copies log list to pv struct for debugging/monitoring

rtyp    �(x)뿓뿓뿓뿓뿓뿓뿬  뿓뿓뿓뿓뿓뿓뿓뿓argument comments뿓뿓뿓뿓뿓뿓뿓뿑븬�  */

UDINT   getSystemUserLogIdent()
{
  return  sysUserEventLog.access.ident;
}

/*————————————————————————————————————————————————————————————————————————————*/

/*————————————————————————————————————————————————————————————————————————————*/
/*! \brief    Points lsvc to a declared memory space
              Declaration is in WBRServicesGlobal.var
              Otherwise, service can use heap memory from wbrMemSvc
    \warning  Must call in Init-SP before calling initLogService() or
              getLogServiceData()

rtyp    �(x)뿓뿓뿓뿓뿓뿓뿓뿓뿓뿓�  뿓뿓뿓뿓뾞rgument comments뿓뿓뿓뿓뿓뿓뿓뿑븬�  */

UDINT   setLogServiceDataAddress(

            wbrLogService_typ * p
          )
{
  lsvc= p;

  return  (UDINT)lsvc;
}

/*————————————————————————————————————————————————————————————————————————————*/

/*! \brief    Init the logging service
*   \pre      Init wbrListService
    \warning  call prior to requestMessageToLog()

rtyp    �(x)뿓뿓뿓뿓뿓�  뿓뿓뿓뿓뿓뿓뿓뿓뿓뾞rgument comments뿓뿓뿓뿓뿓뿓뿓뿑븬�  */

DINT    initLogService()
{
  lsvc->log.str.sLength=    128;
  lsvc->log.str.elements=   128;
  lsvc->log.str.i.maxNodes= 200;

  logList=  (linkedList_typ *)listSvcRequestList(sizeof(wbrLogServiceLogListNode_typ),  lsQUEUE);
  // logList=  (linkedList_typ *)listSvcRequestList(sizeof(wbrLogServiceEventListNode_typ),  lsQUEUE);
  lsvc->log.str.list=  (linkedList_typ *)listSvcRequestList(lsvc->log.str.sLength,  lsQUEUE);

  wbrsnprintf(  sysUserEventLog.access.name
              , sizeof(sysUserEventLog.access.name)
              , "$arlogusr"                              //  System user logbook
              );
  getEventLogInfo(&sysUserEventLog);

  return  0;
}

/** \todo  document * /
rtyp    �(x)뿓뿓뿓뿓뿓뿓뿓뿓뿓뿓뿓뿓뿓뿓뿓�  argument comments뿓뿓뿓뿓뿓뿓뿓븬븰  */

UDINT   wbrLogServicePrintMessageToTextLog()
{
  return  wbrsnprintf((char *)listSvcRequestListNode(lsvc->log.str.list)
                    , lsvc->log.str.sLength
                    , "%s"
                    , lsvc->message
                   );

}

/** \todo  document * /
rtyp    �(x)뿓뿓뿓뿓뿓뿓뿓뿓뿓뿓뿓�  argument comments뿓뿓뿓뿓뿓뿓뿓뿓뿓뿓뿓븬븰  */

UDINT   wbrLogServiceUpdateTextLog()
{
  return  listSvcCharListToStringArray(
                lsvc->log.str.list
              , &lsvc->log.view[0][0]
              , lsvc->log.str.sLength
              , lsvc->log.str.elements > 128 ? 128 : lsvc->log.str.elements
              , lsvc->log.str.i.offset
              , lsvc->log.str.i.pageOffset
              , lsvc->log.str.i.maxNodes
              , 1
              , ""
             );
}

/*! \brief Get info about a logbook
    \pre

rtyp    �(x)뿓뿓뿓뿓뿓�  뿓뿓뿓뿓뿓뿓뿓뿓뿓뾞rgument comments뿓뿓뿓뿓뿓뿓뿓뿑븬�  */

DINT    getLogbookInfo(

          wbrLogServiceLogbookInfo_typ * logInfo                     //!< see type for details
        )
{
 static AsArLogGetInfo_typ fb;

  fb.enable= 1;
  fb.pName=  (UDINT)logInfo->name;

  AsArLogGetInfo(&fb);

  if(!fb.status)
  {
    logInfo->ident=     fb.ident;
    logInfo->length=    fb.len;
    logInfo->memType=   fb.memType;
    logInfo->index=     fb.actualIndex;
    logInfo->formatVer= fb.FormatVer;
  }

  fb.enable= 0;

  return  logInfo->status=    fb.status;
}

/*! \brief Create a new logbook
    \pre

rtyp  �(x)뿓뿓뿓뿓뿓뿓�  뿓뿓뿓뿓뿓뿓뿓뿓뾞rgument comments뿓뿓뿓뿓뿓뿓뿓뿑븬�  */

DINT    createNewLogbook(

            wbrLogServiceLogbookInfo_typ * logInfo                     //!< see type for details
          )
{
 static AsArLogCreate_typ fb;   //! \todo   allocate fb with MemSvc, e.g. if(!logInfo->fb)  allocmem

  fb.enable=  1;
  fb.pName=  (UDINT)logInfo->name;
  fb.len=     logInfo->length;
  fb.memType= logInfo->memType= arlogUSRROM;

  AsArLogCreate(&fb);

  if(!fb.status)
  {
    logInfo->ident=     fb.ident;
    logInfo->status=    fb.status;
    //! \todo   destroy fb
  }

  fb.enable= 0;

  return  logInfo->status=    fb.status;
}

/*! \brief Request a message to be written to a logbook
    \pre   call initLogService()

rtyp  �(x)뿓뿓뿓뿓뿓뿓뿓뿬  뿓뿓뿓뿓뿓뿓뿓argument comments뿓뿓뿓뿓뿓뿓뿓뿑븬�  */

DINT    requestMessageToLog(

            UDINT msgAdr              //!< address that points to the message text, cast as a 32-bit integer
          , UDINT logIdent            //!< identifier of the logbook
          , UDINT logMsgType          //!< 1==info, 2==warn, 3==err, 0==default
          , UDINT erNum               //!< 50000 thru 59999 are reserved for user defined errors
          , UDINT data                //!< address that points to any binary data to include with msg (zero for no data)
          , UDINT dataLen             //!< length of binary data
          )
{
 wbrLogServiceLogListNode_typ *  node=  (wbrLogServiceLogListNode_typ *)listSvcRequestListNode(logList);
 AsArLogWrite_typ *  fb=  node == 0 ? 0 : &node->fb;    //! \todo   eliminate fb?

  if(node == 0)   {
    wbrsnprintf(lsvc->message
              , sizeof(lsvc->message)
              , "Memory was not allocated"
              );
    return  -1;     //  memory was not allocated
  }

  fb->enable= 1;

  if(logMsgType)
  {
    fb->ident=        logIdent;
    fb->logLevel=     logMsgType;
    fb->errornr=      erNum;
    fb->mem=          data;
    fb->len=          dataLen;
  }
  else    // if the message type is not specified, use default ident, logLevel, errornr, and data (default defined in declaration)
  {
    fb->ident=        arlogBASE_USER_LOG_IDENT;
    fb->logLevel=     arEVENTLOG_SEVERITY_INFO;   //  arlogLEVEL_INFO;
    fb->errornr=      50000;
    fb->mem=          0;
    fb->len=          0;
  }

  wbrsnprintf(node->inMsg, 128, "%s", msgAdr);
  fb->asciiString=  (UDINT)(node->inMsg);

  // AsArLogWrite(&node->fb);
  AsArLogWrite(fb);

  if(fb->status == 0xFFFF)
  {
    lsvc->busy=  1;
    return  fb->status;
  }

  if(fb->status)
  {
    wbrsnprintf(lsvc->message,
                sizeof(lsvc->message),
                "Error number %d occurred when writing to the user log",
                fb->status);
  }
  else  {
  wbrsnprintf(lsvc->message,
              sizeof(lsvc->message),
              "Message logged in one cycle");
  }

  lsvc->busy=  logList->numNodes > 10;         //  if more than 10 nodes accumulate, set busy to have writeMessagesToLog() delete them

  getLogServiceData();

  wbrLogServicePrintMessageToTextLog();
  wbrLogServiceUpdateTextLog();
  return  fb->status;
}   ///���\___/���\___/���\___/���\___/���\___/���\___/���\___/���\___/���\�
/*————————————————————————————————————————————————————————————————————————————*/

/*————————————————————————————————————————————————————————————————————————————*/
/*! \brief    Request an event to be written to a logbook
    \pre      call initLogService()
    \warning  ArEventLogWrite fb is defined as synchronous, but requested event
              will fail to be added to the log if fb is on the stack (thus
              using static heap memory)

rtyp  �(x)뿓뿓뿓뿓뿓뿓뿓뿬  뿓뿓뿓뿓뿓뿓뿓argument comments뿓뿓뿓뿓뿓뿓뿓뿑븬�  */

DINT    requestEventToLog(

            UDINT   objectName        //!< Pointer to name of calling object
          , UDINT   logIdent          //!< identifier of the logbook
          , USINT   evSeverity        //!< 0==success, 1==info (default), 2==warn, 3==err,
          ,  UINT   evFacility        //!< range 0 - 0xF (the rest are reserved)
          ,  UINT   evCode            //!< range 0 - 0xFFFF (all)
          ,  DINT   evID              //!< use this if logging a returned ID, e.g. a fb status, etc.
          , UDINT   originID          //!< RecordID of a linked record, e.g. for a multi-entry message/event
          , UDINT   timestamp         //!< application can supply a pointer to a timestamp, use 0 for generated timestamp
          , UDINT   data              //!< address that points to data to be included with event (zero for no data)
          , UDINT   dataSize          //!< length of binary data
          , USINT   dataFormat        //!< 0==binary, 1==null-term text strings, 2==encoded, 100-150 customer(??)
          )
{
 static ArEventLogWrite_typ fb;

  if(!evID && evCode)
    evID= ArEventLogMakeEventID(evSeverity, evFacility, evCode);

  // evID|=  0x20000000;     //  Make sure customer bit is set

  wbrsnprintf(fb.ObjectID, 37, (char *)objectName);
  fb.Ident=          logIdent;
  fb.EventID=        evID;
  fb.OriginRecordID= originID;
  fb.TimeStamp=      timestamp;
  fb.AddData=        data;
  fb.AddDataSize=    dataSize;
  fb.AddDataFormat=  dataFormat;

  fb.Execute= 1;
  ArEventLogWrite(&fb);

  if(fb.Error)
  {
    wbrsnprintf(lsvc->message,
                sizeof(lsvc->message),
                "Error number %d occurred when writing to the user log",
                fb.StatusID);
  genericLog.write.oRecordID= 0;
  }
  else  {
  wbrsnprintf(lsvc->message,
              sizeof(lsvc->message),
              "Event logged in one cycle");
  genericLog.write.oRecordID= fb.RecordID;
  }

  fb.Execute= 0;
  ArEventLogWrite(&fb);      //  Clear the fb for next use

  return  fb.StatusID;
}   ///���\___/���\___/���\___/���\___/���\___/���\___/���\___/���\___/���\�
/*————————————————————————————————————————————————————————————————————————————*/

/*————————————————————————————————————————————————————————————————————————————*/
/*! \brief Request a message to be written to a logbook at level INFO - no data
    \pre   call initLogService()

rtyp  �(x)뿓뿓뿓뿓뿓뿓뿓뿓뿓뿓뿓뿓뿓뿓뿬  argument comments뿓뿓뿓뿓뿓뿓뿓뿑븬�  */

DINT    requestInfoMsgToLogbookNoData(

            UDINT msgAdr              //!< address that points to the message text, cast as a 32-bit integer
          , UDINT logIdent            //!< identifier of the logbook
          )
{
  return  requestMessageToLog(  msgAdr
                              , logIdent
                              , arlogLEVEL_INFO
                              , 50000                 //!<  \todo   create a library constant for this index value
                              , 0
                              , 0
                              );
}   ///���\___/���\___/���\___/���\___/���\___/���\___/���\___/���\___/���\� */

/*! \brief  Request a message to be written to a logbook using an input struct
            hopefully might reduce verbosity of app code
    \pre   call initLogService()

rtyp  �(x)뿓뿓뿓뿓뿓뿓뿓뿓뿓뿓뿓뿓뿓뿓뿬  argument comments뿓뿓뿓뿓뿓뿓뿓뿑븬�  * /

DINT    requestMessageToLogUsingStruct(

            ??_typ * inputStruct              //!< address that points to a struct containing the arguments
          )
{
  return  requestMessageToLog( msgAdr, 0, 0, 0, 0, 0);                          //!<  writes to arlogusr (user logbook) using default settings
}   */

/*————————————————————————————————————————————————————————————————————————————*/
/*! \brief Request a message to be written to a logbook using default settings
    \pre   call initLogService()

rtyp  �(x)뿓뿓뿓뿓뿓뿓뿓뿓뿓뿓뿓�  뿓뿓뿓뾞rgument comments뿓뿓뿓뿓뿓뿓뿓뿑븬�  */

DINT  requestMessageToLogDefault(

            UDINT msgAdr              //!< address that points to the message text, cast as a 32-bit integer
          )
{
  return  requestMessageToLog( msgAdr, 0, 0, 0, 0, 0);                          //!<  writes to arlogusr (user logbook) using default settings
}
/*————————————————————————————————————————————————————————————————————————————*/

/*————————————————————————————————————————————————————————————————————————————*/
/*! \brief Request an event to be written to a logbook using default settings
    \pre

rtyp  �(x)뿓뿓뿓뿓뿓뿓뿓뿓뿓뿓�  뿓뿓뿓뿓뾞rgument comments뿓뿓뿓뿓뿓뿓뿓뿑븬�  */

DINT  requestEventToLogDefault(

            UDINT   objectName        //!< name of calling object
          , UDINT   logIdent          //!< identifier of the logbook
          ,  DINT   evID              //!< use this if logging a returned ID, e.g. a fb status, etc.
          )
{
  return  requestEventToLog( objectName, logIdent, 1,0,0, evID, 0,0,0,0,0);                          //!<  writes to arlogusr (user logbook) using default settings
}
/*————————————————————————————————————————————————————————————————————————————*/

/*————————————————————————————————————————————————————————————————————————————*/
/*! \brief Request an event success to be written to a logbook
    \pre

rtyp  �(x)뿓뿓뿓뿓뿓뿓뿓뿓뿓뿓�  뿓뿓뿓뿓뿓argument comments뿓뿓뿓뿓뿓뿓뿓뿑븬�  */

DINT  requestSuccessEventToLog(

            UDINT   objectName        //!< name of calling object
          , UDINT   logIdent          //!< identifier of the logbook
          ,  UINT   evFacility        //!< range 0 - 0xF (the rest are reserved)
          ,  UINT   evCode            //!< range 0 - 0xFFFF (all)
          , UDINT   timestamp         //!< application can supply a pointer to a timestamp, use 0 for generated timestamp
          , UDINT   msg               //!< address (cast as UDINT) that points to message to be included with success event (zero for no data)
          , UDINT   msgSize           //!< length of binary data
          )

/* Implementation */
{
  // return  requestEventToLog( objectName, logIdent, 0,0,0, evID, 0,0,0,0,0);                          //!<  writes to arlogusr (user logbook) using default settings
  return  requestEventToLog(  objectName
                            , logIdent
                            , arEVENTLOG_SEVERITY_SUCCESS
                            , evFacility
                            , evCode
                            , 0
                            , 0
                            , timestamp
                            , msg
                            , msgSize
                            , arEVENTLOG_ADDFORMAT_TEXT
                            );
}
/*————————————————————————————————————————————————————————————————————————————*/

/*————————————————————————————————————————————————————————————————————————————*/
/*! \brief Request an event to be written to a logbook using default settings
    \pre

rtyp    �(x)뿓뿓뿓뿓뿓뿓뿓뿓뿓뿓뿓�  뿓뿓뿓뾞rgument comments뿓뿓뿓뿓뿓뿓뿓뿑븬�  */

DINT    requestEventToLogUsingObject(

            wbrLogServiceEventLog_typ * el        //!< an event log object
          )
{
  return  requestEventToLog(  el->record.objectName
                            , el->access.ident
                            , 0, 0, 0
                            , el->record.eventID
                            , el->record.originID
                            , el->record.timestamp
                            , el->record.addData
                            , el->record.addDataSize
                            , el->record.addDataFormat
                            );
}
/*————————————————————————————————————————————————————————————————————————————*/

/*————————————————————————————————————————————————————————————————————————————*/
/*! \brief Print the name of the memory type used for logbook storage
    \pre

rtyp  �(x)뿓뿓뿓뿓뿓뿓뿓뿓뿓뿓뿓뿓뿓�  뿓뾞rgument comments뿓뿓뿓뿓뿓뿓뿓뿑븬�  */

static const char *  printMemoryTypeFromPersistence(

            USINT                       persist       //!< 0==Volatile, 1==USRRAM, 2==USRROM.  Use ArEventLog constants in code.
          )
//************************************************
{
  switch(persist)
  {
   case arEVENTLOG_PERSISTENCE_VOLATILE:
    return  "DRAM";
   case arEVENTLOG_PERSISTENCE_REMANENT:
    return  "USRRAM";
   case arEVENTLOG_PERSISTENCE_PERSIST:
    return  "USRROM";
  }

  return  "Ooops! Persistence apparently not in range";
}
/*————————————————————————————————————————————————————————————————————————————*/

/*————————————————————————————————————————————————————————————————————————————*/
/*! \brief Create a new event logbook
    \pre

rtyp  �(x)뿓뿓뿓뿓뿓뿓뿓뿓뿬  뿓뿓뿓뿓뿓뿓argument comments뿓뿓뿓뿓뿓뿓뿓뿑븬�  */

DINT    createNewEventLogbook(

            wbrLogServiceEventLog_typ * logInfo   //!< event log object
          , UDINT                       size      //!< see type for details
          , UDINT                       info      //!< FUTURE, always zero until implemented
          , USINT                       persist   //!< 0==Volatile, 1==USRRAM, 2==USRROM.  Use ArEventLog constants in code.
          )
{
 #define  cNEL_BUF_LEN  128
 static ArEventLogCreate_typ fb;   //! \todo   allocate fb with MemSvc, e.g. if(!logInfo->fb)  allocmem
 static char
                errfmt[cNEL_BUF_LEN - 48]=  "Error %d from facility %d (code %d) when creating event logbook %s."
          ,     fmt[cNEL_BUF_LEN - 48]=     "Event logbook %s of size 0x%X created in %s."
          ,     msg[cNEL_BUF_LEN]=          ""
          ,     len
          ;

  if(!logInfo->busy)   {
    logInfo->done=  logInfo->error=  0;
    wbrsnprintf(fb.Name, sizeof(fb.Name), logInfo->access.name);
    fb.Size=        size;
    fb.Persistence= persist;   //  = arlogUSRROM;    arEVENTLOG_PERSISTENCE_PERSIST
    fb.Info=        0;    //  FUTURE  info;
    fb.Execute= 1;
  }

  ArEventLogCreate(&fb);

  if((logInfo->busy= fb.Busy))      return  logInfo->status;
  if(!(logInfo->error= fb.Error))   logInfo->access.ident= fb.Ident;

  logInfo->done=    fb.Done;
  logInfo->status=  fb.StatusID;

    fb.Execute= 0;
    ArEventLogCreate(&fb);      //  Clear the fb for next use

  //  write success event to log    return  requestCreateSuccessEventToLogUsingObject(logInfo);
  if(!logInfo->error){
    len=  wbrsnprintf(msg
                    , cNEL_BUF_LEN
                    , fmt
                    , logInfo->access.name
                    , size
                    , printMemoryTypeFromPersistence(persist)
                    );
    memset(msg + len + 1, 0, cNEL_BUF_LEN - len - 1);   //  buffer must be flushed
    return  requestEventToLog(  (UDINT)"wbrLogSvc->createNewEventLogbook()"
                              , logInfo->access.ident
                              , 0, 0, 50000
                              , 0
                              , 0
                              , 0
                              , (UDINT)msg
                              , cNEL_BUF_LEN
                              , arEVENTLOG_ADDFORMAT_TEXT
                              );
  }

  decodeEventID(logInfo->status, &eventID);
  len=  wbrsnprintf(msg
                  , cNEL_BUF_LEN
                  , errfmt
                  , eventID.code
                  , eventID.facility
                  , logInfo->status
                  , logInfo->access.name
                  );
  memset(msg + len + 1, 0, cNEL_BUF_LEN - len - 1);
  requestEventToLog(  (UDINT)"wbrLogSvc->createNewEventLogbook()"
                    , sysUserEventLog.access.ident
                    , arEVENTLOG_SEVERITY_ERROR
                    , 0
                    , 50000
                    , 0
                    , 0
                    , 0
                    , (UDINT)msg
                    , cNEL_BUF_LEN
                    , arEVENTLOG_ADDFORMAT_TEXT
                    );
  return  logInfo->status;
}
/*————————————————————————————————————————————————————————————————————————————*/

/* ****************************************************************************/
/*! \brief Request a message to be written to a logbook using default settings
    \pre   call initLogService()

rtyp  �(x)뿓뿓뿓뿓뿓뿓뿓�  뿓뿓뿓뿓뿓뿓뿓뿓뾞rgument comments뿓뿓뿓뿓뿓뿓뿓뿑븬�  */

DINT  writeMessagesToLog()            /// call cyclicly while status is not 0

{
 UDINT  i= logList->numNodes > 100 ? 100 : logList->numNodes;       //  attempt to process all nodes but limit to 100

 wbrLogServiceLogListNode_typ*  node= (wbrLogServiceLogListNode_typ *)listSvcGetHeadData(logList);              //  will assign the address of the data or zero if the list is empty
 // AsArLogWrite_typ *  fb=  &node->fb;    // ! \todo   eliminate fb?
 AsArLogWrite_typ *  fb=  node == 0 ? 0 : &node->fb;    //! \todo   eliminate fb?

  if(!node)
  {
    lsvc->busy=  0;
    wbrsnprintf(lsvc->message,
                sizeof(lsvc->message),
                "No messages to write to a log");
    wbrLogServicePrintMessageToTextLog();
    wbrLogServiceUpdateTextLog();
    getLogServiceData();
    return  -1;
  }

  if(logList->numNodes > lsvc->maxNodesUsed)  lsvc->maxNodesUsed= logList->numNodes;

  for( ; i>0; i--)
  {
    switch(fb->status)
    {
     case 65535:  break;                                                        // busy

     default:                                                                   // error - fall through to 'done'
      wbrsnprintf(lsvc->message,
                  sizeof(lsvc->message),
                  "Error number %d occurred when writing to the user log",
                  fb->status);
      wbrLogServicePrintMessageToTextLog();
      // break;

     case 0:                                                                    // done
      if(listSvcDeleteCurrentNode(logList)) {
        wbrsnprintf(lsvc->message,
                    sizeof(lsvc->message),
                    "Error when freeing node memory");
        wbrLogServicePrintMessageToTextLog();
      }

      if(!(node= (wbrLogServiceLogListNode_typ *)listSvcGetHeadData(logList)))
      {
        lsvc->busy=  0;
        wbrsnprintf(lsvc->message,
                    sizeof(lsvc->message),
                    "All queued messages written to logs");
        wbrLogServicePrintMessageToTextLog();
        wbrLogServiceUpdateTextLog();
        getLogServiceData();
        return  0;
      }
      fb=  &node->fb;
      continue;
    }

    AsArLogWrite(fb);                                                           // call again if busy or error
  }

  wbrLogServiceUpdateTextLog();
  getLogServiceData();
  return  fb->status;
}
/*————————————————————————————————————————————————————————————————————————————*/
```

### Library Logical/UserLibraries/wbrServices/bglibasWBR (ANSIC) - Modified by WBR beginning 2015-01-13

#### bglibasWBR.typ
```iecst
(********************************************************************
 * COPYRIGHT -- belgor
 ********************************************************************
 * Library: bglibas
 * File: bglibas.typ
 * Author: admin
 * Created: March 07, 2012
 ********************************************************************
 * Data types of library bglibas
 ********************************************************************)

TYPE
	BGWBR_TIMER_CONSTANT :
		( (*Included to support legacy bgTimer.h constants*)
		BG_TIMERTIME_1SEC := 1000,
		BG_TIMERTIME_1MIN := 60000,
		BG_TIMERTIME_1HOUR := 3600000
		);
	BGSSM_CONST_XYZ :
		(
		BGSSM_FLAG_COUNT := 5,
		BGSSM_EVENT_COUNT := 5,
		BGSSM_COUNTER_COUNT := 5,
		BGSSM_TIMER_COUNT := 5,
		BGSSM_REGISTER_COUNT := 5,
		BGSSM_SUBROUTINE_COUNT := 5,
		BGSSM_MAX_LOG_ENTRY_INDEX := 31,
		BGSSM_LOG_ENTRIES,
		BGSSM_TEXT_LENGTH := 31,
		BGSSM_MESSAGE_LENGTH_IEC := 127,
		BGSSM_MESSAGE_LENGTH_C
		);
	bgFIFO_typ : 	STRUCT
		iPtrPushData : UDINT;
		cfgEntrySize : UDINT;
		cfgMaxEntries : UDINT;
		oPtrPullData : UDINT;
		oFIFOCount : UDINT;
		oFIFOFull : UDINT;
		oPushIdx : UDINT;
		oPullIdx : UDINT;
		prvFIFOMemory : UDINT;
	END_STRUCT;
	bgSSMScanLimit_typ : 	STRUCT
		breakpoint : BOOL;
		breakpointPrev : BOOL;
		active : BOOL;
		triggerNextScan : BOOL;
		limit : UDINT;
		count : UDINT;
	END_STRUCT;
	bgSSMMessage_typ : 	STRUCT
		log : STRING[BGSSM_MESSAGE_LENGTH_IEC];
		err : STRING[BGSSM_MESSAGE_LENGTH_IEC];
		sts : STRING[BGSSM_MESSAGE_LENGTH_IEC];
	END_STRUCT;
	bgSSMLog_typ : 	STRUCT
		view : ARRAY[0..BGSSM_MAX_LOG_ENTRY_INDEX]OF STRING[BGSSM_MESSAGE_LENGTH_IEC]; (*View window into the log*)
		str : wbrListSvcStringList_typ;
	END_STRUCT;
	bgSSM_typ : 	STRUCT
		scanLimit : bgSSMScanLimit_typ; (*Limits state machine to the number of scans set in .limit member.  Also supports adding breakpoints to the SM.*)
		log : bgSSMLog_typ;
		state : UDINT;
		stateNext : UDINT;
		stateAfterSubIndex : UDINT; (*Index for stateAfterSub below*)
		stateAfterSub : ARRAY[0..BGSSM_SUBROUTINE_COUNT]OF UDINT; (*State to return to after running one or more states defined as a subroutine.  Array allows for subroutine nesting.*)
		stateRet : UDINT;
		stateOld : UDINT;
		stateText : STRING[BGSSM_TEXT_LENGTH];
		pfunInitState : UDINT; (*WBR:*)
		pfunInterrupt : UDINT; (*WBR:*)
		pfunGetStateName : UDINT;
		pfunCyclicCallback : UDINT;
		stateInit : BOOL;
		error : UDINT;
		errorText : STRING[BGSSM_TEXT_LENGTH];
		message : STRING[BGSSM_MESSAGE_LENGTH_IEC]; (*Preformatted state change text for logging.  Can be used for other purposes, but gets written to upon each stateInit.*)
		msg : bgSSMMessage_typ; (*WBR:*)
		event : ARRAY[0..BGSSM_EVENT_COUNT]OF BOOL;
		flag : ARRAY[0..BGSSM_FLAG_COUNT]OF BOOL;
		counter : ARRAY[0..BGSSM_COUNTER_COUNT]OF UDINT;
		value : ARRAY[0..BGSSM_REGISTER_COUNT]OF UDINT;
		timer_x1ms : ARRAY[0..BGSSM_TIMER_COUNT]OF TON;
		dlytimer_x1ms : TON;
		wdogTimer_x1ms : TON;
		dlyCycles : UDINT;
	END_STRUCT;
END_TYPE
```

#### bglibasWBR.fun
```iecst
(********************************************************************
 * COPYRIGHT -- belgor
 ********************************************************************
 * Library: bglibas
 * File: bglibas.fun
 * Author: admin
 * Created: March 07, 2012
 ********************************************************************
 * Functions and function blocks of library bglibas
 ********************************************************************)
(*=========================================================================*)
(*SUPPORT FOR SIMPLE STATE MACHINE (SSM)*)
(*=========================================================================*)

FUNCTION bgSSMInitWbr : UDINT (*Init state machine. MUST be called once, before any other bgSSM function call.*)
	VAR_INPUT
		p : bgSSM_typ;
		pfunInitState : UDINT;
		pfunInterrupt : UDINT;
		pfunCyclicCallback : UDINT;
	END_VAR
END_FUNCTION

FUNCTION bgSSMInit : UDINT (*Init state machine. MUST be called once, before any other bgSSM function call.*)
	VAR_INPUT
		p : bgSSM_typ;
		pfunGetStateName : UDINT;
		pfunCyclicCallback : UDINT;
	END_VAR
END_FUNCTION

FUNCTION bgSSMCyclic : UDINT (*State machine cyclic operation.*)
	VAR_INPUT
		p : bgSSM_typ;
	END_VAR
END_FUNCTION

FUNCTION bgSSMStateNextWithWatchdog : UDINT (*Set SM next state w. timer delay*)
	VAR_INPUT
		p : bgSSM_typ;
		stateNext : UDINT;
		wdogTimeX1ms : UDINT;
	END_VAR
END_FUNCTION

FUNCTION bgSSMStateNextTimeDelay : UDINT (*Set SM next state w. timer delay*)
	VAR_INPUT
		p : bgSSM_typ;
		stateNext : UDINT;
		timeDelayX1ms : UDINT;
	END_VAR
END_FUNCTION

FUNCTION bgSSMStateNextCycleDelay : UDINT (*Set SM next state w. cycles delay*)
	VAR_INPUT
		p : bgSSM_typ;
		stateNext : UDINT;
		delayCycles : UDINT;
	END_VAR
END_FUNCTION

FUNCTION bgSSMStateAfterSub : UDINT (*WBR:  Set SM next state after running subroutine states.*)
	VAR_INPUT
		p : bgSSM_typ;
		stateAfterSub : UDINT;
	END_VAR
END_FUNCTION

FUNCTION bgSSMReturnFromSub : UDINT (*WBR:  Set SM to stateAfterSub state.*)
	VAR_INPUT
		p : bgSSM_typ;
	END_VAR
END_FUNCTION

FUNCTION bgSSMStateNext : UDINT (*Set SM next state.*)
	VAR_INPUT
		p : bgSSM_typ;
		stateNext : UDINT;
	END_VAR
END_FUNCTION

FUNCTION bgSSMIsStateInit : BOOL (*Check if first scan within the current state.*)
	VAR_INPUT
		p : bgSSM_typ;
	END_VAR
END_FUNCTION

FUNCTION bgSSMPrintLogMessage : UDINT (*Check if first scan within the current state.*)
	VAR_INPUT
		p : bgSSM_typ;
	END_VAR
END_FUNCTION

FUNCTION bgSSMPrintToTextLogIEC : UDINT (*Check if first scan within the current state.*)
	VAR_INPUT
		p : bgSSM_typ;
		message : STRING[BGSSM_MESSAGE_LENGTH_IEC];
	END_VAR
END_FUNCTION

FUNCTION bgSSMPrintLogMessageToLogbook : DINT (*Check if first scan within the current state.*)
	VAR_INPUT
		p : bgSSM_typ;
		logIdent : UDINT;
	END_VAR
END_FUNCTION

FUNCTION bgSSMPrintToLogbookIEC : DINT (*Check if first scan within the current state.*)
	VAR_INPUT
		p : bgSSM_typ;
		message : STRING[BGSSM_MESSAGE_LENGTH_IEC];
		logIdent : UDINT;
	END_VAR
END_FUNCTION

FUNCTION bgSSMIsStateInitWBR : BOOL (*Check if first scan within the current state.*)
	VAR_INPUT
		p : bgSSM_typ;
		stateText : STRING[BGSSM_MESSAGE_LENGTH_IEC];
	END_VAR
END_FUNCTION

FUNCTION bgSSMGetState : UDINT (*Get current SM state*)
	VAR_INPUT
		p : bgSSM_typ;
	END_VAR
END_FUNCTION

FUNCTION bgSSMGetStateText : STRING[32] (*Get current SM state name*)
	VAR_INPUT
		p : bgSSM_typ;
	END_VAR
END_FUNCTION
(*=========================================================================*)
(*SUPPORT FOR FIFOs*)
(*=========================================================================*)

FUNCTION bgFIFOInit : UDINT (*Init simple FIFO. Stores upto (entryTotalCount) number of elements. Elements MUST be of the same size.*)
	VAR_INPUT
		p : bgFIFO_typ;
		entrySize : UDINT;
		entryTotalCount : UDINT;
		pFIFOmem : UDINT;
	END_VAR
END_FUNCTION

FUNCTION bgFIFOPush : UDINT (*Push data to FIFO. Content from pSrc is copied into the available FIFO memory. In case of error return value is != 0*)
	VAR_INPUT
		p : bgFIFO_typ;
		pSrc : UDINT;
		srcSize : UDINT;
	END_VAR
END_FUNCTION

FUNCTION bgFIFOPull : UDINT (*Pull (retrive) data from FIFO. Oldest entry from FIFO memory is copied into the provided pDst space. In case of error return value is != 0*)
	VAR_INPUT
		p : bgFIFO_typ;
		pDst : UDINT;
		dstSize : UDINT;
	END_VAR
END_FUNCTION

FUNCTION bgFIFOGetCount : UDINT (*Get number of entries stored in the FIFO*)
	VAR_INPUT
		p : bgFIFO_typ;
	END_VAR
END_FUNCTION

FUNCTION bgFIFOIsFull : UDINT (*Check if FIFO is full*)
	VAR_INPUT
		p : bgFIFO_typ;
	END_VAR
END_FUNCTION
(*=========================================================================*)
(*Support for TIMERs*)
(*=========================================================================*)
FUNCTION bgTimerOffCyclic : UDINT (*Timer cyclic function. Must be called cyclicly for corret timer operation.*)
	VAR_INPUT
		pTOF : TOF;
	END_VAR
END_FUNCTION

FUNCTION bgTimerCyclic : UDINT (*Timer cyclic function. Must be called cyclicly for corret timer operation.*)
	VAR_INPUT
		pTON : TON;
	END_VAR
END_FUNCTION

FUNCTION bgTimerStart : UDINT (*Start timer for a defined amount of time [ms]. IMPORTANT: function uses TON library call. Same restrictions apply!*)
	VAR_INPUT
		pTON : TON;
		timeoutTimeX1ms : UDINT;
	END_VAR
END_FUNCTION

FUNCTION bgTimerStop : UDINT (*Stop the timer.*)
	VAR_INPUT
		pTON : TON;
	END_VAR
END_FUNCTION

FUNCTION bgTimerIsEnabled : BOOL (*Check if timer is enabled.*)
	VAR_INPUT
		pTON : TON;
	END_VAR
END_FUNCTION

FUNCTION bgTimerIsTimeOut : BOOL (*Check if timer has expired.*)
	VAR_INPUT
		pTON : TON;
	END_VAR
END_FUNCTION

FUNCTION bgTimerTimeElapsed : UDINT (*Retrive the elapsed timer time [ms]*)
	VAR_INPUT
		pTON : TON;
	END_VAR
END_FUNCTION

FUNCTION bgTimerTimeRemaining : UDINT (*Retrive the remainig timer time [ms]*)
	VAR_INPUT
		pTON : TON;
	END_VAR
END_FUNCTION
```

#### wbrFunc.h
```c
/********************************************************************
 * \copyright -- Piedmont Automation
 ********************************************************************
 * Program : bglibasWBR
 * \file :   wbrFunc.h
 * \author : Blanton Radford
 * \date Created: May 15, 2015
 *******************************************************************/

#include <bur/plctypes.h>

UDINT  bgSSMPrintToTextLog(struct bgSSM_typ* p, const char* format, ...);
```
